  PROC DrawPart69()
    MoveL Offs(pOrigin,197.94,316.10,6.00),vTravel,z5,tPen\WObj:=wPaper;
    MoveL Offs(pOrigin,197.94,316.10,0.00),v60,z0,tPen\WObj:=wPaper;
    MoveL Offs(pOrigin,198.79,316.95,0.00),v40,z0,tPen\WObj:=wPaper;
    MoveL Offs(pOrigin,197.94,316.10,0.00),v40,fine,tPen\WObj:=wPaper;
    MoveL Offs(pOrigin,197.94,316.10,6.00),v60,z5,tPen\WObj:=wPaper;
    MoveL Offs(pOrigin,199.64,321.62,6.00),vTravel,z5,tPen\WObj:=wPaper;
    MoveL Offs(pOrigin,199.64,321.62,0.00),v60,z0,tPen\WObj:=wPaper;
    MoveL Offs(pOrigin,200.49,322.48,0.00),v40,z0,tPen\WObj:=wPaper;
    MoveL Offs(pOrigin,199.64,321.62,0.00),v40,fine,tPen\WObj:=wPaper;
    MoveL Offs(pOrigin,199.64,321.62,6.00),v60,z5,tPen\WObj:=wPaper;
    MoveL Offs(pOrigin,203.04,325.02,6.00),vTravel,z5,tPen\WObj:=wPaper;
    MoveL Offs(pOrigin,203.04,325.02,0.00),v60,z0,tPen\WObj:=wPaper;
    MoveL Offs(pOrigin,204.24,325.31,0.00),v40,z0,tPen\WObj:=wPaper;
    MoveL Offs(pOrigin,204.52,326.51,0.00),v40,z0,tPen\WObj:=wPaper;
    MoveL Offs(pOrigin,204.95,327.15,0.00),v40,z0,tPen\WObj:=wPaper;
    MoveL Offs(pOrigin,206.86,327.36,0.00),v40,fine,tPen\WObj:=wPaper;
    MoveL Offs(pOrigin,206.86,327.36,6.00),v60,z5,tPen\WObj:=wPaper;
    MoveL Offs(pOrigin,207.29,328.85,6.00),vTravel,z5,tPen\WObj:=wPaper;
    MoveL Offs(pOrigin,207.29,328.85,0.00),v60,z0,tPen\WObj:=wPaper;
    MoveL Offs(pOrigin,208.14,329.49,0.00),v40,z0,tPen\WObj:=wPaper;
    MoveL Offs(pOrigin,207.29,328.85,0.00),v40,fine,tPen\WObj:=wPaper;
    MoveL Offs(pOrigin,207.29,328.85,6.00),v60,z5,tPen\WObj:=wPaper;
    MoveL Offs(pOrigin,206.01,329.27,6.00),vTravel,z5,tPen\WObj:=wPaper;
    MoveL Offs(pOrigin,206.01,329.27,0.00),v60,z0,tPen\WObj:=wPaper;
    MoveL Offs(pOrigin,207.07,330.34,0.00),v40,z0,tPen\WObj:=wPaper;
    MoveL Offs(pOrigin,206.01,329.27,0.00),v40,z0,tPen\WObj:=wPaper;
    MoveL Offs(pOrigin,205.59,328.64,0.00),v40,z0,tPen\WObj:=wPaper;
    MoveL Offs(pOrigin,205.80,329.06,0.00),v40,z0,tPen\WObj:=wPaper;
    MoveL Offs(pOrigin,205.59,328.64,0.00),v40,fine,tPen\WObj:=wPaper;
    MoveL Offs(pOrigin,205.59,328.64,6.00),v60,z5,tPen\WObj:=wPaper;
    MoveL Offs(pOrigin,205.16,329.91,6.00),vTravel,z5,tPen\WObj:=wPaper;
    MoveL Offs(pOrigin,205.16,329.91,0.00),v60,z0,tPen\WObj:=wPaper;
    MoveL Offs(pOrigin,207.29,332.04,0.00),v40,z0,tPen\WObj:=wPaper;
    MoveL Offs(pOrigin,205.16,329.91,0.00),v40,fine,tPen\WObj:=wPaper;
    MoveL Offs(pOrigin,205.16,329.91,6.00),v60,z5,tPen\WObj:=wPaper;
    MoveL Offs(pOrigin,204.95,327.15,6.00),vTravel,z5,tPen\WObj:=wPaper;
    MoveL Offs(pOrigin,204.95,327.15,0.00),v60,z0,tPen\WObj:=wPaper;
    MoveL Offs(pOrigin,205.38,328.21,0.00),v40,z0,tPen\WObj:=wPaper;
    MoveL Offs(pOrigin,207.07,330.12,0.00),v40,z0,tPen\WObj:=wPaper;
    MoveL Offs(pOrigin,209.41,331.75,0.00),v40,z0,tPen\WObj:=wPaper;
    MoveL Offs(pOrigin,210.90,332.04,0.00),v40,z0,tPen\WObj:=wPaper;
    MoveL Offs(pOrigin,210.69,331.19,0.00),v40,z0,tPen\WObj:=wPaper;
    MoveL Offs(pOrigin,210.90,331.61,0.00),v40,z0,tPen\WObj:=wPaper;
    MoveL Offs(pOrigin,210.69,331.19,0.00),v40,fine,tPen\WObj:=wPaper;
    MoveL Offs(pOrigin,210.69,331.19,6.00),v60,z5,tPen\WObj:=wPaper;
    MoveL Offs(pOrigin,208.56,331.40,6.00),vTravel,z5,tPen\WObj:=wPaper;
    MoveL Offs(pOrigin,208.56,331.40,0.00),v60,z0,tPen\WObj:=wPaper;
    MoveL Offs(pOrigin,208.99,331.61,0.00),v40,z0,tPen\WObj:=wPaper;
    MoveL Offs(pOrigin,208.56,331.40,0.00),v40,z0,tPen\WObj:=wPaper;
    MoveL Offs(pOrigin,207.93,330.98,0.00),v40,z0,tPen\WObj:=wPaper;
    MoveL Offs(pOrigin,208.35,331.19,0.00),v40,z0,tPen\WObj:=wPaper;
    MoveL Offs(pOrigin,207.93,330.98,0.00),v40,fine,tPen\WObj:=wPaper;
    MoveL Offs(pOrigin,207.93,330.98,6.00),v60,z5,tPen\WObj:=wPaper;
    MoveL Offs(pOrigin,208.35,329.70,6.00),vTravel,z5,tPen\WObj:=wPaper;
    MoveL Offs(pOrigin,208.35,329.70,0.00),v60,z0,tPen\WObj:=wPaper;
    MoveL Offs(pOrigin,208.77,330.12,0.00),v40,z0,tPen\WObj:=wPaper;
    MoveL Offs(pOrigin,208.35,329.70,0.00),v40,fine,tPen\WObj:=wPaper;
    MoveL Offs(pOrigin,208.35,329.70,6.00),v60,z5,tPen\WObj:=wPaper;
    MoveL Offs(pOrigin,208.14,332.67,6.00),vTravel,z5,tPen\WObj:=wPaper;
    MoveL Offs(pOrigin,208.14,332.67,0.00),v60,z0,tPen\WObj:=wPaper;
    MoveL Offs(pOrigin,208.56,333.10,0.00),v40,z0,tPen\WObj:=wPaper;
    MoveL Offs(pOrigin,208.14,332.67,0.00),v40,fine,tPen\WObj:=wPaper;
    MoveL Offs(pOrigin,208.14,332.67,6.00),v60,z5,tPen\WObj:=wPaper;
    MoveL Offs(pOrigin,209.20,333.52,6.00),vTravel,z5,tPen\WObj:=wPaper;
    MoveL Offs(pOrigin,209.20,333.52,0.00),v60,z0,tPen\WObj:=wPaper;
    MoveL Offs(pOrigin,209.62,333.74,0.00),v40,z0,tPen\WObj:=wPaper;
    MoveL Offs(pOrigin,209.20,333.52,0.00),v40,fine,tPen\WObj:=wPaper;
    MoveL Offs(pOrigin,209.20,333.52,6.00),v60,z5,tPen\WObj:=wPaper;
    MoveL Offs(pOrigin,210.48,334.16,6.00),vTravel,z5,tPen\WObj:=wPaper;
    MoveL Offs(pOrigin,210.48,334.16,0.00),v60,z0,tPen\WObj:=wPaper;
    MoveL Offs(pOrigin,210.90,334.38,0.00),v40,z0,tPen\WObj:=wPaper;
    MoveL Offs(pOrigin,210.48,334.16,0.00),v40,fine,tPen\WObj:=wPaper;
    MoveL Offs(pOrigin,210.48,334.16,6.00),v60,z5,tPen\WObj:=wPaper;
    MoveL Offs(pOrigin,208.14,312.06,6.00),vTravel,z5,tPen\WObj:=wPaper;
    MoveL Offs(pOrigin,208.14,312.06,0.00),v60,z0,tPen\WObj:=wPaper;
    MoveL Offs(pOrigin,208.56,311.85,0.00),v40,z0,tPen\WObj:=wPaper;
    MoveL Offs(pOrigin,208.14,312.06,0.00),v40,fine,tPen\WObj:=wPaper;
    MoveL Offs(pOrigin,208.14,312.06,6.00),v60,z5,tPen\WObj:=wPaper;
    MoveL Offs(pOrigin,214.30,305.90,6.00),vTravel,z5,tPen\WObj:=wPaper;
    MoveL Offs(pOrigin,214.30,305.90,0.00),v60,z0,tPen\WObj:=wPaper;
    MoveL Offs(pOrigin,214.73,306.54,0.00),v40,z0,tPen\WObj:=wPaper;
    MoveL Offs(pOrigin,216.85,306.96,0.00),v40,z0,tPen\WObj:=wPaper;
    MoveL Offs(pOrigin,216.85,306.54,0.00),v40,z0,tPen\WObj:=wPaper;
    MoveL Offs(pOrigin,215.79,305.05,0.00),v40,z0,tPen\WObj:=wPaper;
    MoveL Offs(pOrigin,214.94,305.12,0.00),v40,z0,tPen\WObj:=wPaper;
    MoveL Offs(pOrigin,214.30,305.90,0.00),v40,fine,tPen\WObj:=wPaper;
    MoveL Offs(pOrigin,214.30,305.90,6.00),v60,z5,tPen\WObj:=wPaper;
    MoveL Offs(pOrigin,220.25,307.81,6.00),vTravel,z5,tPen\WObj:=wPaper;
    MoveL Offs(pOrigin,220.25,307.81,0.00),v60,z0,tPen\WObj:=wPaper;
    MoveL Offs(pOrigin,220.46,308.24,0.00),v40,z0,tPen\WObj:=wPaper;
    MoveL Offs(pOrigin,220.25,307.81,0.00),v40,fine,tPen\WObj:=wPaper;
    MoveL Offs(pOrigin,220.25,307.81,6.00),v60,z5,tPen\WObj:=wPaper;
    MoveL Offs(pOrigin,222.38,310.58,6.00),vTravel,z5,tPen\WObj:=wPaper;
    MoveL Offs(pOrigin,222.38,310.58,0.00),v60,z0,tPen\WObj:=wPaper;
    MoveL Offs(pOrigin,221.52,311.85,0.00),v40,fine,tPen\WObj:=wPaper;
    MoveL Offs(pOrigin,221.52,311.85,6.00),v60,z5,tPen\WObj:=wPaper;
    MoveL Offs(pOrigin,221.31,313.34,6.00),vTravel,z5,tPen\WObj:=wPaper;
    MoveL Offs(pOrigin,221.31,313.34,0.00),v60,z0,tPen\WObj:=wPaper;
    MoveL Offs(pOrigin,221.52,312.27,0.00),v40,z0,tPen\WObj:=wPaper;
    MoveL Offs(pOrigin,221.10,311.92,0.00),v40,z0,tPen\WObj:=wPaper;
    MoveL Offs(pOrigin,220.46,312.13,0.00),v40,z0,tPen\WObj:=wPaper;
    MoveL Offs(pOrigin,219.61,313.34,0.00),v40,fine,tPen\WObj:=wPaper;
    MoveL Offs(pOrigin,219.61,313.34,6.00),v60,z5,tPen\WObj:=wPaper;
    MoveL Offs(pOrigin,209.84,301.01,6.00),vTravel,z5,tPen\WObj:=wPaper;
    MoveL Offs(pOrigin,209.84,301.01,0.00),v60,z0,tPen\WObj:=wPaper;
    MoveL Offs(pOrigin,209.34,298.89,0.00),v40,z0,tPen\WObj:=wPaper;
    MoveL Offs(pOrigin,207.50,296.76,0.00),v40,z0,tPen\WObj:=wPaper;
    MoveL Offs(pOrigin,207.93,296.98,0.00),v40,z0,tPen\WObj:=wPaper;
    MoveL Offs(pOrigin,208.35,297.40,0.00),v40,z0,tPen\WObj:=wPaper;
    MoveL Offs(pOrigin,207.93,296.98,0.00),v40,fine,tPen\WObj:=wPaper;
    MoveL Offs(pOrigin,207.93,296.98,6.00),v60,z5,tPen\WObj:=wPaper;
    MoveL Offs(pOrigin,209.20,266.38,6.00),vTravel,z5,tPen\WObj:=wPaper;
    MoveL Offs(pOrigin,209.20,266.38,0.00),v60,z0,tPen\WObj:=wPaper;
    MoveL Offs(pOrigin,208.14,266.16,0.00),v40,z0,tPen\WObj:=wPaper;
    MoveL Offs(pOrigin,207.50,265.31,0.00),v40,fine,tPen\WObj:=wPaper;
    MoveL Offs(pOrigin,207.50,265.31,6.00),v60,z5,tPen\WObj:=wPaper;
    MoveL Offs(pOrigin,207.29,260.85,6.00),vTravel,z5,tPen\WObj:=wPaper;
    MoveL Offs(pOrigin,207.29,260.85,0.00),v60,z0,tPen\WObj:=wPaper;
    MoveL Offs(pOrigin,207.93,260.00,0.00),v40,z0,tPen\WObj:=wPaper;
    MoveL Offs(pOrigin,207.93,258.94,0.00),v40,z0,tPen\WObj:=wPaper;
  ENDPROC

  PROC DrawPart70()
    MoveL Offs(pOrigin,207.93,258.94,0.00),v40,z0,tPen\WObj:=wPaper;
    MoveL Offs(pOrigin,208.07,258.30,0.00),v40,z0,tPen\WObj:=wPaper;
    MoveL Offs(pOrigin,207.07,257.02,0.00),v40,z0,tPen\WObj:=wPaper;
    MoveL Offs(pOrigin,207.29,251.71,0.00),v40,z0,tPen\WObj:=wPaper;
    MoveL Offs(pOrigin,207.07,248.95,0.00),v40,z0,tPen\WObj:=wPaper;
    MoveL Offs(pOrigin,206.44,248.17,0.00),v40,z0,tPen\WObj:=wPaper;
    MoveL Offs(pOrigin,205.66,248.31,0.00),v40,z0,tPen\WObj:=wPaper;
    MoveL Offs(pOrigin,205.38,250.23,0.00),v40,z0,tPen\WObj:=wPaper;
    MoveL Offs(pOrigin,205.80,250.65,0.00),v40,z0,tPen\WObj:=wPaper;
    MoveL Offs(pOrigin,205.02,250.44,0.00),v40,z0,tPen\WObj:=wPaper;
    MoveL Offs(pOrigin,204.38,252.14,0.00),v40,z0,tPen\WObj:=wPaper;
    MoveL Offs(pOrigin,203.39,257.02,0.00),v40,z0,tPen\WObj:=wPaper;
    MoveL Offs(pOrigin,203.68,258.09,0.00),v40,z0,tPen\WObj:=wPaper;
    MoveL Offs(pOrigin,203.46,259.36,0.00),v40,z0,tPen\WObj:=wPaper;
    MoveL Offs(pOrigin,202.90,260.00,0.00),v40,z0,tPen\WObj:=wPaper;
    MoveL Offs(pOrigin,202.54,261.70,0.00),v40,z0,tPen\WObj:=wPaper;
    MoveL Offs(pOrigin,201.98,261.91,0.00),v40,z0,tPen\WObj:=wPaper;
    MoveL Offs(pOrigin,201.98,261.91,0.00),v40,z0,tPen\WObj:=wPaper;
    MoveL Offs(pOrigin,201.69,260.00,0.00),v40,z0,tPen\WObj:=wPaper;
    MoveL Offs(pOrigin,200.91,259.79,0.00),v40,z0,tPen\WObj:=wPaper;
    MoveL Offs(pOrigin,201.98,259.79,0.00),v40,z0,tPen\WObj:=wPaper;
    MoveL Offs(pOrigin,202.12,258.51,0.00),v40,z0,tPen\WObj:=wPaper;
    MoveL Offs(pOrigin,203.25,257.45,0.00),v40,fine,tPen\WObj:=wPaper;
    MoveL Offs(pOrigin,203.25,257.45,6.00),v60,z5,tPen\WObj:=wPaper;
    MoveL Offs(pOrigin,201.55,256.81,6.00),vTravel,z5,tPen\WObj:=wPaper;
    MoveL Offs(pOrigin,201.55,256.81,0.00),v60,z0,tPen\WObj:=wPaper;
    MoveL Offs(pOrigin,201.12,249.59,0.00),v40,fine,tPen\WObj:=wPaper;
    MoveL Offs(pOrigin,201.12,249.59,6.00),v60,z5,tPen\WObj:=wPaper;
    MoveL Offs(pOrigin,198.57,248.74,6.00),vTravel,z5,tPen\WObj:=wPaper;
    MoveL Offs(pOrigin,198.57,248.74,0.00),v60,z0,tPen\WObj:=wPaper;
    MoveL Offs(pOrigin,198.15,249.38,0.00),v40,z0,tPen\WObj:=wPaper;
    MoveL Offs(pOrigin,198.57,248.74,0.00),v40,fine,tPen\WObj:=wPaper;
    MoveL Offs(pOrigin,198.57,248.74,6.00),v60,z5,tPen\WObj:=wPaper;
    MoveL Offs(pOrigin,197.73,247.68,6.00),vTravel,z5,tPen\WObj:=wPaper;
    MoveL Offs(pOrigin,197.73,247.68,0.00),v60,z0,tPen\WObj:=wPaper;
    MoveL Offs(pOrigin,197.30,248.31,0.00),v40,z0,tPen\WObj:=wPaper;
    MoveL Offs(pOrigin,197.73,247.68,0.00),v40,fine,tPen\WObj:=wPaper;
    MoveL Offs(pOrigin,197.73,247.68,6.00),v60,z5,tPen\WObj:=wPaper;
    MoveL Offs(pOrigin,198.79,245.98,6.00),vTravel,z5,tPen\WObj:=wPaper;
    MoveL Offs(pOrigin,198.79,245.98,0.00),v60,z0,tPen\WObj:=wPaper;
    MoveL Offs(pOrigin,198.36,246.61,0.00),v40,z0,tPen\WObj:=wPaper;
    MoveL Offs(pOrigin,198.79,245.98,0.00),v40,fine,tPen\WObj:=wPaper;
    MoveL Offs(pOrigin,198.79,245.98,6.00),v60,z5,tPen\WObj:=wPaper;
    MoveL Offs(pOrigin,199.64,247.04,6.00),vTravel,z5,tPen\WObj:=wPaper;
    MoveL Offs(pOrigin,199.64,247.04,0.00),v60,z0,tPen\WObj:=wPaper;
    MoveL Offs(pOrigin,199.43,247.46,0.00),v40,z0,tPen\WObj:=wPaper;
    MoveL Offs(pOrigin,199.64,247.04,0.00),v40,fine,tPen\WObj:=wPaper;
    MoveL Offs(pOrigin,199.64,247.04,6.00),v60,z5,tPen\WObj:=wPaper;
    MoveL Offs(pOrigin,197.73,250.01,6.00),vTravel,z5,tPen\WObj:=wPaper;
    MoveL Offs(pOrigin,197.73,250.01,0.00),v60,z0,tPen\WObj:=wPaper;
    MoveL Offs(pOrigin,197.51,250.44,0.00),v40,z0,tPen\WObj:=wPaper;
    MoveL Offs(pOrigin,197.73,250.01,0.00),v40,z0,tPen\WObj:=wPaper;
    MoveL Offs(pOrigin,197.30,250.86,0.00),v40,z0,tPen\WObj:=wPaper;
    MoveL Offs(pOrigin,197.09,251.29,0.00),v40,z0,tPen\WObj:=wPaper;
    MoveL Offs(pOrigin,197.30,250.86,0.00),v40,fine,tPen\WObj:=wPaper;
    MoveL Offs(pOrigin,197.30,250.86,6.00),v60,z5,tPen\WObj:=wPaper;
    MoveL Offs(pOrigin,196.24,249.80,6.00),vTravel,z5,tPen\WObj:=wPaper;
    MoveL Offs(pOrigin,196.24,249.80,0.00),v60,z0,tPen\WObj:=wPaper;
    MoveL Offs(pOrigin,196.02,250.23,0.00),v40,z0,tPen\WObj:=wPaper;
    MoveL Offs(pOrigin,196.24,249.80,0.00),v40,fine,tPen\WObj:=wPaper;
    MoveL Offs(pOrigin,196.24,249.80,6.00),v60,z5,tPen\WObj:=wPaper;
    MoveL Offs(pOrigin,205.59,248.10,6.00),vTravel,z5,tPen\WObj:=wPaper;
    MoveL Offs(pOrigin,205.59,248.10,0.00),v60,z0,tPen\WObj:=wPaper;
    MoveL Offs(pOrigin,204.95,247.04,0.00),v40,z0,tPen\WObj:=wPaper;
    MoveL Offs(pOrigin,204.81,245.34,0.00),v40,z0,tPen\WObj:=wPaper;
    MoveL Offs(pOrigin,205.09,243.85,0.00),v40,z0,tPen\WObj:=wPaper;
    MoveL Offs(pOrigin,205.59,243.21,0.00),v40,z0,tPen\WObj:=wPaper;
    MoveL Offs(pOrigin,205.59,243.21,0.00),v40,z0,tPen\WObj:=wPaper;
    MoveL Offs(pOrigin,205.80,241.94,0.00),v40,z0,tPen\WObj:=wPaper;
    MoveL Offs(pOrigin,206.65,241.51,0.00),v40,z0,tPen\WObj:=wPaper;
    MoveL Offs(pOrigin,206.65,241.51,0.00),v40,z0,tPen\WObj:=wPaper;
    MoveL Offs(pOrigin,206.86,242.79,0.00),v40,z0,tPen\WObj:=wPaper;
    MoveL Offs(pOrigin,206.44,243.21,0.00),v40,z0,tPen\WObj:=wPaper;
    MoveL Offs(pOrigin,206.44,243.21,0.00),v40,z0,tPen\WObj:=wPaper;
    MoveL Offs(pOrigin,206.86,245.98,0.00),v40,z0,tPen\WObj:=wPaper;
    MoveL Offs(pOrigin,206.65,248.10,0.00),v40,fine,tPen\WObj:=wPaper;
    MoveL Offs(pOrigin,206.65,248.10,6.00),v60,z5,tPen\WObj:=wPaper;
    MoveL Offs(pOrigin,207.29,257.24,6.00),vTravel,z5,tPen\WObj:=wPaper;
    MoveL Offs(pOrigin,207.29,257.24,0.00),v60,z0,tPen\WObj:=wPaper;
    MoveL Offs(pOrigin,207.71,257.45,0.00),v40,z0,tPen\WObj:=wPaper;
    MoveL Offs(pOrigin,208.07,257.24,0.00),v40,z0,tPen\WObj:=wPaper;
    MoveL Offs(pOrigin,209.34,253.41,0.00),v40,z0,tPen\WObj:=wPaper;
    MoveL Offs(pOrigin,210.90,251.07,0.00),v40,z0,tPen\WObj:=wPaper;
    MoveL Offs(pOrigin,211.96,250.30,0.00),v40,z0,tPen\WObj:=wPaper;
    MoveL Offs(pOrigin,214.94,249.59,0.00),v40,z0,tPen\WObj:=wPaper;
    MoveL Offs(pOrigin,223.65,249.80,0.00),v40,z0,tPen\WObj:=wPaper;
    MoveL Offs(pOrigin,230.45,251.07,0.00),v40,z0,tPen\WObj:=wPaper;
    MoveL Offs(pOrigin,232.79,251.85,0.00),v40,z0,tPen\WObj:=wPaper;
    MoveL Offs(pOrigin,234.91,253.62,0.00),v40,z0,tPen\WObj:=wPaper;
    MoveL Offs(pOrigin,235.55,254.90,0.00),v40,fine,tPen\WObj:=wPaper;
    MoveL Offs(pOrigin,235.55,254.90,6.00),v60,z5,tPen\WObj:=wPaper;
    MoveL Offs(pOrigin,236.19,256.39,6.00),vTravel,z5,tPen\WObj:=wPaper;
    MoveL Offs(pOrigin,236.19,256.39,0.00),v60,z0,tPen\WObj:=wPaper;
    MoveL Offs(pOrigin,236.19,257.24,0.00),v40,z0,tPen\WObj:=wPaper;
    MoveL Offs(pOrigin,236.82,257.88,0.00),v40,z0,tPen\WObj:=wPaper;
    MoveL Offs(pOrigin,236.82,257.88,0.00),v40,z0,tPen\WObj:=wPaper;
    MoveL Offs(pOrigin,237.68,257.02,0.00),v40,z0,tPen\WObj:=wPaper;
    MoveL Offs(pOrigin,237.60,256.17,0.00),v40,z0,tPen\WObj:=wPaper;
    MoveL Offs(pOrigin,237.04,255.75,0.00),v40,z0,tPen\WObj:=wPaper;
    MoveL Offs(pOrigin,237.04,255.75,0.00),v40,z0,tPen\WObj:=wPaper;
    MoveL Offs(pOrigin,236.19,256.39,0.00),v40,z0,tPen\WObj:=wPaper;
    MoveL Offs(pOrigin,236.19,256.39,0.00),v40,z0,tPen\WObj:=wPaper;
    MoveL Offs(pOrigin,235.69,255.96,0.00),v40,z0,tPen\WObj:=wPaper;
    MoveL Offs(pOrigin,235.62,255.11,0.00),v40,z0,tPen\WObj:=wPaper;
    MoveL Offs(pOrigin,236.40,255.18,0.00),v40,z0,tPen\WObj:=wPaper;
    MoveL Offs(pOrigin,237.04,255.75,0.00),v40,fine,tPen\WObj:=wPaper;
    MoveL Offs(pOrigin,237.04,255.75,6.00),v60,z5,tPen\WObj:=wPaper;
    MoveL Offs(pOrigin,236.82,259.58,6.00),vTravel,z5,tPen\WObj:=wPaper;
    MoveL Offs(pOrigin,236.82,259.58,0.00),v60,z0,tPen\WObj:=wPaper;
    MoveL Offs(pOrigin,236.75,258.51,0.00),v40,z0,tPen\WObj:=wPaper;
    MoveL Offs(pOrigin,235.98,258.09,0.00),v40,z0,tPen\WObj:=wPaper;
    MoveL Offs(pOrigin,234.49,259.58,0.00),v40,z0,tPen\WObj:=wPaper;
    MoveL Offs(pOrigin,234.49,259.58,0.00),v40,z0,tPen\WObj:=wPaper;
    MoveL Offs(pOrigin,235.12,260.21,0.00),v40,z0,tPen\WObj:=wPaper;
    MoveL Offs(pOrigin,235.12,260.21,0.00),v40,z0,tPen\WObj:=wPaper;
    MoveL Offs(pOrigin,235.12,260.00,0.00),v40,z0,tPen\WObj:=wPaper;
    MoveL Offs(pOrigin,236.19,260.21,0.00),v40,z0,tPen\WObj:=wPaper;
    MoveL Offs(pOrigin,236.82,259.58,0.00),v40,z0,tPen\WObj:=wPaper;
    MoveL Offs(pOrigin,236.82,259.58,0.00),v40,z0,tPen\WObj:=wPaper;
    MoveL Offs(pOrigin,237.04,260.85,0.00),v40,z0,tPen\WObj:=wPaper;
  ENDPROC

  PROC DrawPart71()
    MoveL Offs(pOrigin,237.04,260.85,0.00),v40,z0,tPen\WObj:=wPaper;
    MoveL Offs(pOrigin,238.31,262.12,0.00),v40,z0,tPen\WObj:=wPaper;
    MoveL Offs(pOrigin,238.24,262.98,0.00),v40,z0,tPen\WObj:=wPaper;
    MoveL Offs(pOrigin,237.25,263.83,0.00),v40,z0,tPen\WObj:=wPaper;
    MoveL Offs(pOrigin,237.25,263.83,0.00),v40,z0,tPen\WObj:=wPaper;
    MoveL Offs(pOrigin,238.10,265.31,0.00),v40,z0,tPen\WObj:=wPaper;
    MoveL Offs(pOrigin,240.23,266.16,0.00),v40,z0,tPen\WObj:=wPaper;
    MoveL Offs(pOrigin,243.41,266.38,0.00),v40,z0,tPen\WObj:=wPaper;
    MoveL Offs(pOrigin,244.69,266.16,0.00),v40,fine,tPen\WObj:=wPaper;
    MoveL Offs(pOrigin,244.69,266.16,6.00),v60,z5,tPen\WObj:=wPaper;
    MoveL Offs(pOrigin,244.69,267.86,6.00),vTravel,z5,tPen\WObj:=wPaper;
    MoveL Offs(pOrigin,244.69,267.86,0.00),v60,z0,tPen\WObj:=wPaper;
    MoveL Offs(pOrigin,245.75,267.65,0.00),v40,z0,tPen\WObj:=wPaper;
    MoveL Offs(pOrigin,245.75,267.86,0.00),v40,z0,tPen\WObj:=wPaper;
    MoveL Offs(pOrigin,246.60,267.86,0.00),v40,z0,tPen\WObj:=wPaper;
    MoveL Offs(pOrigin,245.96,267.93,0.00),v40,z0,tPen\WObj:=wPaper;
    MoveL Offs(pOrigin,245.75,268.50,0.00),v40,z0,tPen\WObj:=wPaper;
    MoveL Offs(pOrigin,246.81,269.14,0.00),v40,fine,tPen\WObj:=wPaper;
    MoveL Offs(pOrigin,246.81,269.14,6.00),v60,z5,tPen\WObj:=wPaper;
    MoveL Offs(pOrigin,247.24,270.41,6.00),vTravel,z5,tPen\WObj:=wPaper;
    MoveL Offs(pOrigin,247.24,270.41,0.00),v60,z0,tPen\WObj:=wPaper;
    MoveL Offs(pOrigin,248.73,270.62,0.00),v40,fine,tPen\WObj:=wPaper;
    MoveL Offs(pOrigin,248.73,270.62,6.00),v60,z5,tPen\WObj:=wPaper;
    MoveL Offs(pOrigin,247.24,270.41,6.00),vTravel,z5,tPen\WObj:=wPaper;
    MoveL Offs(pOrigin,247.24,270.41,0.00),v60,z0,tPen\WObj:=wPaper;
    MoveL Offs(pOrigin,246.18,271.90,0.00),v40,z0,tPen\WObj:=wPaper;
    MoveL Offs(pOrigin,246.25,272.54,0.00),v40,z0,tPen\WObj:=wPaper;
    MoveL Offs(pOrigin,246.81,272.96,0.00),v40,fine,tPen\WObj:=wPaper;
    MoveL Offs(pOrigin,246.81,272.96,6.00),v60,z5,tPen\WObj:=wPaper;
    MoveL Offs(pOrigin,245.11,270.20,6.00),vTravel,z5,tPen\WObj:=wPaper;
    MoveL Offs(pOrigin,245.11,270.20,0.00),v60,z0,tPen\WObj:=wPaper;
    MoveL Offs(pOrigin,243.98,271.26,0.00),v40,z0,tPen\WObj:=wPaper;
    MoveL Offs(pOrigin,243.13,273.17,0.00),v40,z0,tPen\WObj:=wPaper;
    MoveL Offs(pOrigin,242.14,277.64,0.00),v40,fine,tPen\WObj:=wPaper;
    MoveL Offs(pOrigin,242.14,277.64,6.00),v60,z5,tPen\WObj:=wPaper;
    MoveL Offs(pOrigin,237.46,267.01,6.00),vTravel,z5,tPen\WObj:=wPaper;
    MoveL Offs(pOrigin,237.46,267.01,0.00),v60,z0,tPen\WObj:=wPaper;
    MoveL Offs(pOrigin,237.04,266.23,0.00),v40,z0,tPen\WObj:=wPaper;
    MoveL Offs(pOrigin,236.40,266.23,0.00),v40,z0,tPen\WObj:=wPaper;
    MoveL Offs(pOrigin,235.69,267.01,0.00),v40,z0,tPen\WObj:=wPaper;
    MoveL Offs(pOrigin,236.40,267.44,0.00),v40,fine,tPen\WObj:=wPaper;
    MoveL Offs(pOrigin,236.40,267.44,6.00),v60,z5,tPen\WObj:=wPaper;
    MoveL Offs(pOrigin,235.34,265.52,6.00),vTravel,z5,tPen\WObj:=wPaper;
    MoveL Offs(pOrigin,235.34,265.52,0.00),v60,z0,tPen\WObj:=wPaper;
    MoveL Offs(pOrigin,235.98,264.67,0.00),v40,z0,tPen\WObj:=wPaper;
    MoveL Offs(pOrigin,237.25,263.83,0.00),v40,z0,tPen\WObj:=wPaper;
    MoveL Offs(pOrigin,236.82,263.83,0.00),v40,z0,tPen\WObj:=wPaper;
    MoveL Offs(pOrigin,236.19,262.55,0.00),v40,z0,tPen\WObj:=wPaper;
    MoveL Offs(pOrigin,235.34,262.34,0.00),v40,z0,tPen\WObj:=wPaper;
    MoveL Offs(pOrigin,235.34,262.34,0.00),v40,z0,tPen\WObj:=wPaper;
    MoveL Offs(pOrigin,234.91,261.27,0.00),v40,z0,tPen\WObj:=wPaper;
    MoveL Offs(pOrigin,235.12,260.21,0.00),v40,z0,tPen\WObj:=wPaper;
    MoveL Offs(pOrigin,234.49,259.58,0.00),v40,z0,tPen\WObj:=wPaper;
    MoveL Offs(pOrigin,233.21,259.50,0.00),v40,z0,tPen\WObj:=wPaper;
    MoveL Offs(pOrigin,232.72,258.09,0.00),v40,z0,tPen\WObj:=wPaper;
    MoveL Offs(pOrigin,231.30,256.60,0.00),v40,z0,tPen\WObj:=wPaper;
    MoveL Offs(pOrigin,227.05,254.26,0.00),v40,fine,tPen\WObj:=wPaper;
    MoveL Offs(pOrigin,227.05,254.26,6.00),v60,z5,tPen\WObj:=wPaper;
    MoveL Offs(pOrigin,226.41,259.15,6.00),vTravel,z5,tPen\WObj:=wPaper;
    MoveL Offs(pOrigin,226.41,259.15,0.00),v60,z0,tPen\WObj:=wPaper;
    MoveL Offs(pOrigin,223.65,258.94,0.00),v40,z0,tPen\WObj:=wPaper;
    MoveL Offs(pOrigin,223.23,259.15,0.00),v40,z0,tPen\WObj:=wPaper;
    MoveL Offs(pOrigin,222.87,260.00,0.00),v40,z0,tPen\WObj:=wPaper;
    MoveL Offs(pOrigin,224.07,260.85,0.00),v40,z0,tPen\WObj:=wPaper;
    MoveL Offs(pOrigin,224.07,260.85,0.00),v40,z0,tPen\WObj:=wPaper;
    MoveL Offs(pOrigin,224.29,261.49,0.00),v40,z0,tPen\WObj:=wPaper;
    MoveL Offs(pOrigin,224.71,261.70,0.00),v40,z0,tPen\WObj:=wPaper;
    MoveL Offs(pOrigin,225.56,261.63,0.00),v40,z0,tPen\WObj:=wPaper;
    MoveL Offs(pOrigin,226.20,261.06,0.00),v40,z0,tPen\WObj:=wPaper;
    MoveL Offs(pOrigin,227.05,261.06,0.00),v40,z0,tPen\WObj:=wPaper;
    MoveL Offs(pOrigin,227.48,260.64,0.00),v40,z0,tPen\WObj:=wPaper;
    MoveL Offs(pOrigin,228.32,260.64,0.00),v40,z0,tPen\WObj:=wPaper;
    MoveL Offs(pOrigin,228.96,261.27,0.00),v40,z0,tPen\WObj:=wPaper;
    MoveL Offs(pOrigin,228.96,261.91,0.00),v40,z0,tPen\WObj:=wPaper;
    MoveL Offs(pOrigin,229.03,261.49,0.00),v40,z0,tPen\WObj:=wPaper;
    MoveL Offs(pOrigin,229.60,261.27,0.00),v40,z0,tPen\WObj:=wPaper;
    MoveL Offs(pOrigin,230.88,261.63,0.00),v40,z0,tPen\WObj:=wPaper;
    MoveL Offs(pOrigin,231.51,262.34,0.00),v40,z0,tPen\WObj:=wPaper;
    MoveL Offs(pOrigin,231.30,261.70,0.00),v40,z0,tPen\WObj:=wPaper;
    MoveL Offs(pOrigin,232.36,261.27,0.00),v40,z0,tPen\WObj:=wPaper;
    MoveL Offs(pOrigin,233.21,261.49,0.00),v40,z0,tPen\WObj:=wPaper;
    MoveL Offs(pOrigin,233.21,261.49,0.00),v40,z0,tPen\WObj:=wPaper;
    MoveL Offs(pOrigin,234.91,261.49,0.00),v40,fine,tPen\WObj:=wPaper;
    MoveL Offs(pOrigin,234.91,261.49,6.00),v60,z5,tPen\WObj:=wPaper;
    MoveL Offs(pOrigin,236.19,262.34,6.00),vTravel,z5,tPen\WObj:=wPaper;
    MoveL Offs(pOrigin,236.19,262.34,0.00),v60,z0,tPen\WObj:=wPaper;
    MoveL Offs(pOrigin,237.04,260.85,0.00),v40,fine,tPen\WObj:=wPaper;
    MoveL Offs(pOrigin,237.04,260.85,6.00),v60,z5,tPen\WObj:=wPaper;
    MoveL Offs(pOrigin,233.00,259.58,6.00),vTravel,z5,tPen\WObj:=wPaper;
    MoveL Offs(pOrigin,233.00,259.58,0.00),v60,z0,tPen\WObj:=wPaper;
    MoveL Offs(pOrigin,231.51,259.29,0.00),v40,z0,tPen\WObj:=wPaper;
    MoveL Offs(pOrigin,227.26,257.31,0.00),v40,z0,tPen\WObj:=wPaper;
    MoveL Offs(pOrigin,224.50,256.60,0.00),v40,z0,tPen\WObj:=wPaper;
    MoveL Offs(pOrigin,223.23,256.60,0.00),v40,z0,tPen\WObj:=wPaper;
    MoveL Offs(pOrigin,222.16,255.96,0.00),v40,fine,tPen\WObj:=wPaper;
    MoveL Offs(pOrigin,222.16,255.96,6.00),v60,z5,tPen\WObj:=wPaper;
    MoveL Offs(pOrigin,221.74,257.24,6.00),vTravel,z5,tPen\WObj:=wPaper;
    MoveL Offs(pOrigin,221.74,257.24,0.00),v60,z0,tPen\WObj:=wPaper;
    MoveL Offs(pOrigin,219.19,257.45,0.00),v40,fine,tPen\WObj:=wPaper;
    MoveL Offs(pOrigin,219.19,257.45,6.00),v60,z5,tPen\WObj:=wPaper;
    MoveL Offs(pOrigin,213.24,263.40,6.00),vTravel,z5,tPen\WObj:=wPaper;
    MoveL Offs(pOrigin,213.24,263.40,0.00),v60,z0,tPen\WObj:=wPaper;
    MoveL Offs(pOrigin,213.10,264.89,0.00),v40,z0,tPen\WObj:=wPaper;
    MoveL Offs(pOrigin,214.51,266.59,0.00),v40,z0,tPen\WObj:=wPaper;
    MoveL Offs(pOrigin,219.19,267.86,0.00),v40,z0,tPen\WObj:=wPaper;
    MoveL Offs(pOrigin,219.19,267.86,0.00),v40,z0,tPen\WObj:=wPaper;
    MoveL Offs(pOrigin,220.89,268.08,0.00),v40,z0,tPen\WObj:=wPaper;
    MoveL Offs(pOrigin,221.74,267.86,0.00),v40,fine,tPen\WObj:=wPaper;
    MoveL Offs(pOrigin,221.74,267.86,6.00),v60,z5,tPen\WObj:=wPaper;
    MoveL Offs(pOrigin,233.21,267.44,6.00),vTravel,z5,tPen\WObj:=wPaper;
    MoveL Offs(pOrigin,233.21,267.44,0.00),v60,z0,tPen\WObj:=wPaper;
    MoveL Offs(pOrigin,233.85,268.08,0.00),v40,fine,tPen\WObj:=wPaper;
    MoveL Offs(pOrigin,233.85,268.08,6.00),v60,z5,tPen\WObj:=wPaper;
    MoveL Offs(pOrigin,252.12,268.29,6.00),vTravel,z5,tPen\WObj:=wPaper;
    MoveL Offs(pOrigin,252.12,268.29,0.00),v60,z0,tPen\WObj:=wPaper;
    MoveL Offs(pOrigin,252.55,268.71,0.00),v40,z0,tPen\WObj:=wPaper;
    MoveL Offs(pOrigin,252.12,268.29,0.00),v40,fine,tPen\WObj:=wPaper;
    MoveL Offs(pOrigin,252.12,268.29,6.00),v60,z5,tPen\WObj:=wPaper;
    MoveL Offs(pOrigin,255.95,269.35,6.00),vTravel,z5,tPen\WObj:=wPaper;
    MoveL Offs(pOrigin,255.95,269.35,0.00),v60,z0,tPen\WObj:=wPaper;
  ENDPROC

  PROC DrawPart72()
    MoveL Offs(pOrigin,257.44,269.99,0.00),v40,z0,tPen\WObj:=wPaper;
    MoveL Offs(pOrigin,259.14,269.77,0.00),v40,fine,tPen\WObj:=wPaper;
    MoveL Offs(pOrigin,259.14,269.77,6.00),v60,z5,tPen\WObj:=wPaper;
    MoveL Offs(pOrigin,276.35,263.83,6.00),vTravel,z5,tPen\WObj:=wPaper;
    MoveL Offs(pOrigin,276.35,263.83,0.00),v60,z0,tPen\WObj:=wPaper;
    MoveL Offs(pOrigin,275.92,263.40,0.00),v40,z0,tPen\WObj:=wPaper;
    MoveL Offs(pOrigin,276.14,262.34,0.00),v40,z0,tPen\WObj:=wPaper;
    MoveL Offs(pOrigin,276.14,261.91,0.00),v40,z0,tPen\WObj:=wPaper;
    MoveL Offs(pOrigin,275.71,261.49,0.00),v40,z0,tPen\WObj:=wPaper;
    MoveL Offs(pOrigin,275.92,260.64,0.00),v40,fine,tPen\WObj:=wPaper;
    MoveL Offs(pOrigin,275.92,260.64,6.00),v60,z5,tPen\WObj:=wPaper;
    MoveL Offs(pOrigin,279.75,272.75,6.00),vTravel,z5,tPen\WObj:=wPaper;
    MoveL Offs(pOrigin,279.75,272.75,0.00),v60,z0,tPen\WObj:=wPaper;
    MoveL Offs(pOrigin,280.39,273.17,0.00),v40,z0,tPen\WObj:=wPaper;
    MoveL Offs(pOrigin,282.09,273.17,0.00),v40,fine,tPen\WObj:=wPaper;
    MoveL Offs(pOrigin,282.09,273.17,6.00),v60,z5,tPen\WObj:=wPaper;
    MoveL Offs(pOrigin,280.39,279.12,6.00),vTravel,z5,tPen\WObj:=wPaper;
    MoveL Offs(pOrigin,280.39,279.12,0.00),v60,z0,tPen\WObj:=wPaper;
    MoveL Offs(pOrigin,279.61,279.41,0.00),v40,z0,tPen\WObj:=wPaper;
    MoveL Offs(pOrigin,279.33,280.19,0.00),v40,z0,tPen\WObj:=wPaper;
    MoveL Offs(pOrigin,279.96,280.83,0.00),v40,fine,tPen\WObj:=wPaper;
    MoveL Offs(pOrigin,279.96,280.83,6.00),v60,z5,tPen\WObj:=wPaper;
    MoveL Offs(pOrigin,291.44,271.48,6.00),vTravel,z5,tPen\WObj:=wPaper;
    MoveL Offs(pOrigin,291.44,271.48,0.00),v60,z0,tPen\WObj:=wPaper;
    MoveL Offs(pOrigin,291.44,270.41,0.00),v40,z0,tPen\WObj:=wPaper;
    MoveL Offs(pOrigin,290.38,269.99,0.00),v40,z0,tPen\WObj:=wPaper;
    MoveL Offs(pOrigin,290.38,269.99,0.00),v40,z0,tPen\WObj:=wPaper;
    MoveL Offs(pOrigin,290.16,269.42,0.00),v40,z0,tPen\WObj:=wPaper;
    MoveL Offs(pOrigin,289.10,268.92,0.00),v40,z0,tPen\WObj:=wPaper;
    MoveL Offs(pOrigin,289.17,268.36,0.00),v40,z0,tPen\WObj:=wPaper;
    MoveL Offs(pOrigin,289.95,268.29,0.00),v40,z0,tPen\WObj:=wPaper;
    MoveL Offs(pOrigin,289.95,268.29,0.00),v40,z0,tPen\WObj:=wPaper;
    MoveL Offs(pOrigin,290.38,269.35,0.00),v40,z0,tPen\WObj:=wPaper;
    MoveL Offs(pOrigin,290.38,269.99,0.00),v40,z0,tPen\WObj:=wPaper;
    MoveL Offs(pOrigin,290.16,270.41,0.00),v40,z0,tPen\WObj:=wPaper;
    MoveL Offs(pOrigin,290.38,271.05,0.00),v40,z0,tPen\WObj:=wPaper;
    MoveL Offs(pOrigin,291.44,271.48,0.00),v40,fine,tPen\WObj:=wPaper;
    MoveL Offs(pOrigin,291.44,271.48,6.00),v60,z5,tPen\WObj:=wPaper;
    MoveL Offs(pOrigin,293.56,269.77,6.00),vTravel,z5,tPen\WObj:=wPaper;
    MoveL Offs(pOrigin,293.56,269.77,0.00),v60,z0,tPen\WObj:=wPaper;
    MoveL Offs(pOrigin,294.20,270.41,0.00),v40,z0,tPen\WObj:=wPaper;
    MoveL Offs(pOrigin,293.56,269.77,0.00),v40,fine,tPen\WObj:=wPaper;
    MoveL Offs(pOrigin,293.56,269.77,6.00),v60,z5,tPen\WObj:=wPaper;
    MoveL Offs(pOrigin,290.80,267.23,6.00),vTravel,z5,tPen\WObj:=wPaper;
    MoveL Offs(pOrigin,290.80,267.23,0.00),v60,z0,tPen\WObj:=wPaper;
    MoveL Offs(pOrigin,289.95,267.86,0.00),v40,z0,tPen\WObj:=wPaper;
    MoveL Offs(pOrigin,289.95,268.29,0.00),v40,fine,tPen\WObj:=wPaper;
    MoveL Offs(pOrigin,289.95,268.29,6.00),v60,z5,tPen\WObj:=wPaper;
    MoveL Offs(pOrigin,264.66,312.27,6.00),vTravel,z5,tPen\WObj:=wPaper;
    MoveL Offs(pOrigin,264.66,312.27,0.00),v60,z0,tPen\WObj:=wPaper;
    MoveL Offs(pOrigin,264.45,312.49,0.00),v40,z0,tPen\WObj:=wPaper;
    MoveL Offs(pOrigin,263.60,312.27,0.00),v40,z0,tPen\WObj:=wPaper;
    MoveL Offs(pOrigin,263.60,312.27,0.00),v40,z0,tPen\WObj:=wPaper;
    MoveL Offs(pOrigin,259.14,311.21,0.00),v40,z0,tPen\WObj:=wPaper;
    MoveL Offs(pOrigin,259.14,311.21,0.00),v40,z0,tPen\WObj:=wPaper;
    MoveL Offs(pOrigin,259.77,313.12,0.00),v40,fine,tPen\WObj:=wPaper;
    MoveL Offs(pOrigin,259.77,313.12,6.00),v60,z5,tPen\WObj:=wPaper;
    MoveL Offs(pOrigin,258.29,312.27,6.00),vTravel,z5,tPen\WObj:=wPaper;
    MoveL Offs(pOrigin,258.29,312.27,0.00),v60,z0,tPen\WObj:=wPaper;
    MoveL Offs(pOrigin,258.71,312.70,0.00),v40,z0,tPen\WObj:=wPaper;
    MoveL Offs(pOrigin,258.29,312.27,0.00),v40,fine,tPen\WObj:=wPaper;
    MoveL Offs(pOrigin,258.29,312.27,6.00),v60,z5,tPen\WObj:=wPaper;
    MoveL Offs(pOrigin,256.59,310.79,6.00),vTravel,z5,tPen\WObj:=wPaper;
    MoveL Offs(pOrigin,256.59,310.79,0.00),v60,z0,tPen\WObj:=wPaper;
    MoveL Offs(pOrigin,257.01,311.42,0.00),v40,z0,tPen\WObj:=wPaper;
    MoveL Offs(pOrigin,256.59,310.79,0.00),v40,fine,tPen\WObj:=wPaper;
    MoveL Offs(pOrigin,256.59,310.79,6.00),v60,z5,tPen\WObj:=wPaper;
    MoveL Offs(pOrigin,255.52,313.55,6.00),vTravel,z5,tPen\WObj:=wPaper;
    MoveL Offs(pOrigin,255.52,313.55,0.00),v60,z0,tPen\WObj:=wPaper;
    MoveL Offs(pOrigin,255.95,313.98,0.00),v40,z0,tPen\WObj:=wPaper;
    MoveL Offs(pOrigin,255.52,313.55,0.00),v40,fine,tPen\WObj:=wPaper;
    MoveL Offs(pOrigin,255.52,313.55,6.00),v60,z5,tPen\WObj:=wPaper;
    MoveL Offs(pOrigin,253.19,313.98,6.00),vTravel,z5,tPen\WObj:=wPaper;
    MoveL Offs(pOrigin,253.19,313.98,0.00),v60,z0,tPen\WObj:=wPaper;
    MoveL Offs(pOrigin,253.82,314.61,0.00),v40,z0,tPen\WObj:=wPaper;
    MoveL Offs(pOrigin,253.19,313.98,0.00),v40,fine,tPen\WObj:=wPaper;
    MoveL Offs(pOrigin,253.19,313.98,6.00),v60,z5,tPen\WObj:=wPaper;
    MoveL Offs(pOrigin,252.55,312.49,6.00),vTravel,z5,tPen\WObj:=wPaper;
    MoveL Offs(pOrigin,252.55,312.49,0.00),v60,z0,tPen\WObj:=wPaper;
    MoveL Offs(pOrigin,252.98,313.55,0.00),v40,z0,tPen\WObj:=wPaper;
    MoveL Offs(pOrigin,254.82,315.67,0.00),v40,z0,tPen\WObj:=wPaper;
    MoveL Offs(pOrigin,255.31,318.01,0.00),v40,z0,tPen\WObj:=wPaper;
    MoveL Offs(pOrigin,256.16,318.44,0.00),v40,z0,tPen\WObj:=wPaper;
    MoveL Offs(pOrigin,256.66,320.14,0.00),v40,z0,tPen\WObj:=wPaper;
    MoveL Offs(pOrigin,257.65,320.99,0.00),v40,z0,tPen\WObj:=wPaper;
    MoveL Offs(pOrigin,258.71,321.20,0.00),v40,z0,tPen\WObj:=wPaper;
    MoveL Offs(pOrigin,259.35,321.84,0.00),v40,z0,tPen\WObj:=wPaper;
    MoveL Offs(pOrigin,258.71,321.20,0.00),v40,fine,tPen\WObj:=wPaper;
    MoveL Offs(pOrigin,258.71,321.20,6.00),v60,z5,tPen\WObj:=wPaper;
    MoveL Offs(pOrigin,252.12,319.08,6.00),vTravel,z5,tPen\WObj:=wPaper;
    MoveL Offs(pOrigin,252.12,319.08,0.00),v60,z0,tPen\WObj:=wPaper;
    MoveL Offs(pOrigin,249.79,318.65,0.00),v40,z0,tPen\WObj:=wPaper;
    MoveL Offs(pOrigin,248.94,319.08,0.00),v40,z0,tPen\WObj:=wPaper;
    MoveL Offs(pOrigin,247.45,318.86,0.00),v40,fine,tPen\WObj:=wPaper;
    MoveL Offs(pOrigin,247.45,318.86,6.00),v60,z5,tPen\WObj:=wPaper;
    MoveL Offs(pOrigin,246.60,321.20,6.00),vTravel,z5,tPen\WObj:=wPaper;
    MoveL Offs(pOrigin,246.60,321.20,0.00),v60,z0,tPen\WObj:=wPaper;
    MoveL Offs(pOrigin,247.02,321.41,0.00),v40,z0,tPen\WObj:=wPaper;
    MoveL Offs(pOrigin,246.60,321.20,0.00),v40,fine,tPen\WObj:=wPaper;
    MoveL Offs(pOrigin,246.60,321.20,6.00),v60,z5,tPen\WObj:=wPaper;
    MoveL Offs(pOrigin,244.69,319.92,6.00),vTravel,z5,tPen\WObj:=wPaper;
    MoveL Offs(pOrigin,244.69,319.92,0.00),v60,z0,tPen\WObj:=wPaper;
    MoveL Offs(pOrigin,245.54,320.70,0.00),v40,z0,tPen\WObj:=wPaper;
    MoveL Offs(pOrigin,247.24,321.41,0.00),v40,z0,tPen\WObj:=wPaper;
    MoveL Offs(pOrigin,248.73,323.47,0.00),v40,z0,tPen\WObj:=wPaper;
    MoveL Offs(pOrigin,250.43,324.17,0.00),v40,z0,tPen\WObj:=wPaper;
    MoveL Offs(pOrigin,252.27,326.16,0.00),v40,z0,tPen\WObj:=wPaper;
    MoveL Offs(pOrigin,252.55,329.06,0.00),v40,z0,tPen\WObj:=wPaper;
    MoveL Offs(pOrigin,251.77,331.19,0.00),v40,z0,tPen\WObj:=wPaper;
    MoveL Offs(pOrigin,250.85,331.61,0.00),v40,z0,tPen\WObj:=wPaper;
    MoveL Offs(pOrigin,250.85,331.61,0.00),v40,z0,tPen\WObj:=wPaper;
    MoveL Offs(pOrigin,250.43,332.67,0.00),v40,z0,tPen\WObj:=wPaper;
    MoveL Offs(pOrigin,249.15,333.52,0.00),v40,z0,tPen\WObj:=wPaper;
    MoveL Offs(pOrigin,249.15,333.95,0.00),v40,z0,tPen\WObj:=wPaper;
    MoveL Offs(pOrigin,247.45,334.23,0.00),v40,z0,tPen\WObj:=wPaper;
    MoveL Offs(pOrigin,246.39,335.23,0.00),v40,z0,tPen\WObj:=wPaper;
    MoveL Offs(pOrigin,247.02,334.59,0.00),v40,z0,tPen\WObj:=wPaper;
    MoveL Offs(pOrigin,246.81,335.01,0.00),v40,z0,tPen\WObj:=wPaper;
    MoveL Offs(pOrigin,247.02,334.59,0.00),v40,fine,tPen\WObj:=wPaper;
    MoveL Offs(pOrigin,247.02,334.59,6.00),v60,z5,tPen\WObj:=wPaper;
  ENDPROC

  PROC DrawPart73()
    MoveL Offs(pOrigin,247.66,336.29,6.00),vTravel,z5,tPen\WObj:=wPaper;
    MoveL Offs(pOrigin,247.66,336.29,0.00),v60,z0,tPen\WObj:=wPaper;
    MoveL Offs(pOrigin,248.09,336.08,0.00),v40,z0,tPen\WObj:=wPaper;
    MoveL Offs(pOrigin,247.66,336.29,0.00),v40,z0,tPen\WObj:=wPaper;
    MoveL Offs(pOrigin,247.24,336.50,0.00),v40,z0,tPen\WObj:=wPaper;
    MoveL Offs(pOrigin,248.65,335.65,0.00),v40,z0,tPen\WObj:=wPaper;
    MoveL Offs(pOrigin,249.15,334.59,0.00),v40,fine,tPen\WObj:=wPaper;
    MoveL Offs(pOrigin,249.15,334.59,6.00),v60,z5,tPen\WObj:=wPaper;
    MoveL Offs(pOrigin,250.64,334.38,6.00),vTravel,z5,tPen\WObj:=wPaper;
    MoveL Offs(pOrigin,250.64,334.38,0.00),v60,z0,tPen\WObj:=wPaper;
    MoveL Offs(pOrigin,250.85,333.95,0.00),v40,z0,tPen\WObj:=wPaper;
    MoveL Offs(pOrigin,250.64,334.38,0.00),v40,z0,tPen\WObj:=wPaper;
    MoveL Offs(pOrigin,251.27,333.74,0.00),v40,z0,tPen\WObj:=wPaper;
    MoveL Offs(pOrigin,251.49,333.31,0.00),v40,z0,tPen\WObj:=wPaper;
    MoveL Offs(pOrigin,251.27,333.74,0.00),v40,z0,tPen\WObj:=wPaper;
    MoveL Offs(pOrigin,251.91,333.10,0.00),v40,z0,tPen\WObj:=wPaper;
    MoveL Offs(pOrigin,252.12,332.67,0.00),v40,z0,tPen\WObj:=wPaper;
    MoveL Offs(pOrigin,251.91,333.10,0.00),v40,fine,tPen\WObj:=wPaper;
    MoveL Offs(pOrigin,251.91,333.10,6.00),v60,z5,tPen\WObj:=wPaper;
    MoveL Offs(pOrigin,252.34,334.80,6.00),vTravel,z5,tPen\WObj:=wPaper;
    MoveL Offs(pOrigin,252.34,334.80,0.00),v60,z0,tPen\WObj:=wPaper;
    MoveL Offs(pOrigin,254.60,332.46,0.00),v40,z0,tPen\WObj:=wPaper;
    MoveL Offs(pOrigin,255.31,330.76,0.00),v40,fine,tPen\WObj:=wPaper;
    MoveL Offs(pOrigin,255.31,330.76,6.00),v60,z5,tPen\WObj:=wPaper;
    MoveL Offs(pOrigin,250.85,331.61,6.00),vTravel,z5,tPen\WObj:=wPaper;
    MoveL Offs(pOrigin,250.85,331.61,0.00),v60,z0,tPen\WObj:=wPaper;
    MoveL Offs(pOrigin,251.06,328.64,0.00),v40,z0,tPen\WObj:=wPaper;
    MoveL Offs(pOrigin,250.43,326.09,0.00),v40,z0,tPen\WObj:=wPaper;
    MoveL Offs(pOrigin,250.85,325.02,0.00),v40,fine,tPen\WObj:=wPaper;
    MoveL Offs(pOrigin,250.85,325.02,6.00),v60,z5,tPen\WObj:=wPaper;
    MoveL Offs(pOrigin,246.39,323.96,6.00),vTravel,z5,tPen\WObj:=wPaper;
    MoveL Offs(pOrigin,246.39,323.96,0.00),v60,z0,tPen\WObj:=wPaper;
    MoveL Offs(pOrigin,247.66,327.58,0.00),v40,z0,tPen\WObj:=wPaper;
    MoveL Offs(pOrigin,247.66,330.55,0.00),v40,z0,tPen\WObj:=wPaper;
    MoveL Offs(pOrigin,246.67,333.10,0.00),v40,z0,tPen\WObj:=wPaper;
    MoveL Offs(pOrigin,245.96,333.52,0.00),v40,z0,tPen\WObj:=wPaper;
    MoveL Offs(pOrigin,245.11,333.52,0.00),v40,z0,tPen\WObj:=wPaper;
    MoveL Offs(pOrigin,245.11,333.52,0.00),v40,z0,tPen\WObj:=wPaper;
    MoveL Offs(pOrigin,244.05,335.01,0.00),v40,z0,tPen\WObj:=wPaper;
    MoveL Offs(pOrigin,244.05,335.65,0.00),v40,z0,tPen\WObj:=wPaper;
    MoveL Offs(pOrigin,243.20,336.08,0.00),v40,z0,tPen\WObj:=wPaper;
    MoveL Offs(pOrigin,242.99,335.65,0.00),v40,z0,tPen\WObj:=wPaper;
    MoveL Offs(pOrigin,241.50,335.65,0.00),v40,fine,tPen\WObj:=wPaper;
    MoveL Offs(pOrigin,241.50,335.65,6.00),v60,z5,tPen\WObj:=wPaper;
    MoveL Offs(pOrigin,242.14,334.59,6.00),vTravel,z5,tPen\WObj:=wPaper;
    MoveL Offs(pOrigin,242.14,334.59,0.00),v60,z0,tPen\WObj:=wPaper;
    MoveL Offs(pOrigin,242.35,334.16,0.00),v40,z0,tPen\WObj:=wPaper;
    MoveL Offs(pOrigin,242.14,334.59,0.00),v40,z0,tPen\WObj:=wPaper;
    MoveL Offs(pOrigin,242.77,333.95,0.00),v40,z0,tPen\WObj:=wPaper;
    MoveL Offs(pOrigin,242.99,333.52,0.00),v40,z0,tPen\WObj:=wPaper;
    MoveL Offs(pOrigin,242.77,333.95,0.00),v40,z0,tPen\WObj:=wPaper;
    MoveL Offs(pOrigin,243.41,333.10,0.00),v40,z0,tPen\WObj:=wPaper;
    MoveL Offs(pOrigin,243.62,332.67,0.00),v40,z0,tPen\WObj:=wPaper;
    MoveL Offs(pOrigin,243.41,333.10,0.00),v40,fine,tPen\WObj:=wPaper;
    MoveL Offs(pOrigin,243.41,333.10,6.00),v60,z5,tPen\WObj:=wPaper;
    MoveL Offs(pOrigin,245.54,335.65,6.00),vTravel,z5,tPen\WObj:=wPaper;
    MoveL Offs(pOrigin,245.54,335.65,0.00),v60,z0,tPen\WObj:=wPaper;
    MoveL Offs(pOrigin,245.82,335.51,0.00),v40,z0,tPen\WObj:=wPaper;
    MoveL Offs(pOrigin,244.90,336.00,0.00),v40,z0,tPen\WObj:=wPaper;
    MoveL Offs(pOrigin,243.84,335.79,0.00),v40,z0,tPen\WObj:=wPaper;
    MoveL Offs(pOrigin,242.77,336.85,0.00),v40,z0,tPen\WObj:=wPaper;
    MoveL Offs(pOrigin,240.01,337.99,0.00),v40,z0,tPen\WObj:=wPaper;
    MoveL Offs(pOrigin,237.25,338.62,0.00),v40,z0,tPen\WObj:=wPaper;
    MoveL Offs(pOrigin,236.40,338.41,0.00),v40,fine,tPen\WObj:=wPaper;
    MoveL Offs(pOrigin,236.40,338.41,6.00),v60,z5,tPen\WObj:=wPaper;
    MoveL Offs(pOrigin,244.05,338.41,6.00),vTravel,z5,tPen\WObj:=wPaper;
    MoveL Offs(pOrigin,244.05,338.41,0.00),v60,z0,tPen\WObj:=wPaper;
    MoveL Offs(pOrigin,245.32,338.62,0.00),v40,z0,tPen\WObj:=wPaper;
    MoveL Offs(pOrigin,245.32,338.62,0.00),v40,z0,tPen\WObj:=wPaper;
    MoveL Offs(pOrigin,245.32,338.84,0.00),v40,z0,tPen\WObj:=wPaper;
    MoveL Offs(pOrigin,246.39,338.62,0.00),v40,z0,tPen\WObj:=wPaper;
    MoveL Offs(pOrigin,246.39,337.99,0.00),v40,z0,tPen\WObj:=wPaper;
    MoveL Offs(pOrigin,246.39,338.41,0.00),v40,z0,tPen\WObj:=wPaper;
    MoveL Offs(pOrigin,247.02,338.62,0.00),v40,z0,tPen\WObj:=wPaper;
    MoveL Offs(pOrigin,247.45,337.99,0.00),v40,z0,tPen\WObj:=wPaper;
    MoveL Offs(pOrigin,247.45,337.99,0.00),v40,z0,tPen\WObj:=wPaper;
    MoveL Offs(pOrigin,250.21,337.77,0.00),v40,z0,tPen\WObj:=wPaper;
    MoveL Offs(pOrigin,252.55,337.14,0.00),v40,fine,tPen\WObj:=wPaper;
    MoveL Offs(pOrigin,252.55,337.14,6.00),v60,z5,tPen\WObj:=wPaper;
    MoveL Offs(pOrigin,252.98,335.86,6.00),vTravel,z5,tPen\WObj:=wPaper;
    MoveL Offs(pOrigin,252.98,335.86,0.00),v60,z0,tPen\WObj:=wPaper;
    MoveL Offs(pOrigin,252.62,336.92,0.00),v40,z0,tPen\WObj:=wPaper;
    MoveL Offs(pOrigin,254.04,337.14,0.00),v40,z0,tPen\WObj:=wPaper;
    MoveL Offs(pOrigin,254.04,337.14,0.00),v40,z0,tPen\WObj:=wPaper;
    MoveL Offs(pOrigin,254.89,337.63,0.00),v40,z0,tPen\WObj:=wPaper;
    MoveL Offs(pOrigin,257.65,336.29,0.00),v40,fine,tPen\WObj:=wPaper;
    MoveL Offs(pOrigin,257.65,336.29,6.00),v60,z5,tPen\WObj:=wPaper;
    MoveL Offs(pOrigin,254.68,336.08,6.00),vTravel,z5,tPen\WObj:=wPaper;
    MoveL Offs(pOrigin,254.68,336.08,0.00),v60,z0,tPen\WObj:=wPaper;
    MoveL Offs(pOrigin,255.52,335.65,0.00),v40,z0,tPen\WObj:=wPaper;
    MoveL Offs(pOrigin,255.95,334.45,0.00),v40,z0,tPen\WObj:=wPaper;
    MoveL Offs(pOrigin,255.10,334.52,0.00),v40,z0,tPen\WObj:=wPaper;
    MoveL Offs(pOrigin,254.25,335.44,0.00),v40,z0,tPen\WObj:=wPaper;
    MoveL Offs(pOrigin,254.25,335.44,0.00),v40,z0,tPen\WObj:=wPaper;
    MoveL Offs(pOrigin,253.61,335.44,0.00),v40,z0,tPen\WObj:=wPaper;
    MoveL Offs(pOrigin,253.40,335.86,0.00),v40,z0,tPen\WObj:=wPaper;
    MoveL Offs(pOrigin,253.61,335.65,0.00),v40,z0,tPen\WObj:=wPaper;
    MoveL Offs(pOrigin,254.68,336.08,0.00),v40,z0,tPen\WObj:=wPaper;
    MoveL Offs(pOrigin,254.04,337.14,0.00),v40,fine,tPen\WObj:=wPaper;
    MoveL Offs(pOrigin,254.04,337.14,6.00),v60,z5,tPen\WObj:=wPaper;
    MoveL Offs(pOrigin,247.45,337.99,6.00),vTravel,z5,tPen\WObj:=wPaper;
    MoveL Offs(pOrigin,247.45,337.99,0.00),v60,z0,tPen\WObj:=wPaper;
    MoveL Offs(pOrigin,247.45,337.77,0.00),v40,z0,tPen\WObj:=wPaper;
    MoveL Offs(pOrigin,246.39,337.99,0.00),v40,z0,tPen\WObj:=wPaper;
    MoveL Offs(pOrigin,246.39,337.99,0.00),v40,z0,tPen\WObj:=wPaper;
    MoveL Offs(pOrigin,245.75,337.99,0.00),v40,z0,tPen\WObj:=wPaper;
    MoveL Offs(pOrigin,245.32,338.62,0.00),v40,fine,tPen\WObj:=wPaper;
    MoveL Offs(pOrigin,245.32,338.62,6.00),v60,z5,tPen\WObj:=wPaper;
    MoveL Offs(pOrigin,244.05,338.41,6.00),vTravel,z5,tPen\WObj:=wPaper;
    MoveL Offs(pOrigin,244.05,338.41,0.00),v60,z0,tPen\WObj:=wPaper;
    MoveL Offs(pOrigin,244.26,337.77,0.00),v40,z0,tPen\WObj:=wPaper;
    MoveL Offs(pOrigin,246.60,336.71,0.00),v40,fine,tPen\WObj:=wPaper;
    MoveL Offs(pOrigin,246.60,336.71,6.00),v60,z5,tPen\WObj:=wPaper;
    MoveL Offs(pOrigin,238.10,321.84,6.00),vTravel,z5,tPen\WObj:=wPaper;
    MoveL Offs(pOrigin,238.10,321.84,0.00),v60,z0,tPen\WObj:=wPaper;
    MoveL Offs(pOrigin,237.04,320.77,0.00),v40,fine,tPen\WObj:=wPaper;
    MoveL Offs(pOrigin,237.04,320.77,6.00),v60,z5,tPen\WObj:=wPaper;
    MoveL Offs(pOrigin,240.44,320.14,6.00),vTravel,z5,tPen\WObj:=wPaper;
    MoveL Offs(pOrigin,240.44,320.14,0.00),v60,z0,tPen\WObj:=wPaper;
    MoveL Offs(pOrigin,241.29,320.99,0.00),v40,z0,tPen\WObj:=wPaper;
  ENDPROC

  PROC DrawPart74()
    MoveL Offs(pOrigin,240.44,320.14,0.00),v40,fine,tPen\WObj:=wPaper;
    MoveL Offs(pOrigin,240.44,320.14,6.00),v60,z5,tPen\WObj:=wPaper;
    MoveL Offs(pOrigin,238.74,317.59,6.00),vTravel,z5,tPen\WObj:=wPaper;
    MoveL Offs(pOrigin,238.74,317.59,0.00),v60,z0,tPen\WObj:=wPaper;
    MoveL Offs(pOrigin,238.31,313.34,0.00),v40,z0,tPen\WObj:=wPaper;
    MoveL Offs(pOrigin,238.67,312.06,0.00),v40,z0,tPen\WObj:=wPaper;
    MoveL Offs(pOrigin,239.59,311.42,0.00),v40,fine,tPen\WObj:=wPaper;
    MoveL Offs(pOrigin,239.59,311.42,6.00),v60,z5,tPen\WObj:=wPaper;
    MoveL Offs(pOrigin,238.74,310.15,6.00),vTravel,z5,tPen\WObj:=wPaper;
    MoveL Offs(pOrigin,238.74,310.15,0.00),v60,z0,tPen\WObj:=wPaper;
    MoveL Offs(pOrigin,238.17,310.36,0.00),v40,z0,tPen\WObj:=wPaper;
    MoveL Offs(pOrigin,237.25,312.06,0.00),v40,z0,tPen\WObj:=wPaper;
    MoveL Offs(pOrigin,237.25,312.06,0.00),v40,z0,tPen\WObj:=wPaper;
    MoveL Offs(pOrigin,236.68,312.49,0.00),v40,z0,tPen\WObj:=wPaper;
    MoveL Offs(pOrigin,236.33,314.19,0.00),v40,z0,tPen\WObj:=wPaper;
    MoveL Offs(pOrigin,235.98,314.40,0.00),v40,fine,tPen\WObj:=wPaper;
    MoveL Offs(pOrigin,235.98,314.40,6.00),v60,z5,tPen\WObj:=wPaper;
    MoveL Offs(pOrigin,237.25,312.06,6.00),vTravel,z5,tPen\WObj:=wPaper;
    MoveL Offs(pOrigin,237.25,312.06,0.00),v60,z0,tPen\WObj:=wPaper;
    MoveL Offs(pOrigin,237.46,312.49,0.00),v40,z0,tPen\WObj:=wPaper;
    MoveL Offs(pOrigin,237.25,314.83,0.00),v40,z0,tPen\WObj:=wPaper;
    MoveL Offs(pOrigin,237.68,316.95,0.00),v40,fine,tPen\WObj:=wPaper;
    MoveL Offs(pOrigin,237.68,316.95,6.00),v60,z5,tPen\WObj:=wPaper;
    MoveL Offs(pOrigin,240.01,316.10,6.00),vTravel,z5,tPen\WObj:=wPaper;
    MoveL Offs(pOrigin,240.01,316.10,0.00),v60,z0,tPen\WObj:=wPaper;
    MoveL Offs(pOrigin,240.23,316.52,0.00),v40,z0,tPen\WObj:=wPaper;
    MoveL Offs(pOrigin,240.01,316.10,0.00),v40,fine,tPen\WObj:=wPaper;
    MoveL Offs(pOrigin,240.01,316.10,6.00),v60,z5,tPen\WObj:=wPaper;
    MoveL Offs(pOrigin,206.23,260.85,6.00),vTravel,z5,tPen\WObj:=wPaper;
    MoveL Offs(pOrigin,206.23,260.85,0.00),v60,z0,tPen\WObj:=wPaper;
    MoveL Offs(pOrigin,206.01,261.27,0.00),v40,z0,tPen\WObj:=wPaper;
    MoveL Offs(pOrigin,206.23,260.85,0.00),v40,fine,tPen\WObj:=wPaper;
    MoveL Offs(pOrigin,206.23,260.85,6.00),v60,z5,tPen\WObj:=wPaper;
    MoveL Offs(pOrigin,207.93,258.94,6.00),vTravel,z5,tPen\WObj:=wPaper;
    MoveL Offs(pOrigin,207.93,258.94,0.00),v60,z0,tPen\WObj:=wPaper;
    MoveL Offs(pOrigin,207.07,258.73,0.00),v40,z0,tPen\WObj:=wPaper;
    MoveL Offs(pOrigin,207.29,257.88,0.00),v40,z0,tPen\WObj:=wPaper;
    MoveL Offs(pOrigin,207.07,257.88,0.00),v40,z0,tPen\WObj:=wPaper;
    MoveL Offs(pOrigin,207.71,257.66,0.00),v40,z0,tPen\WObj:=wPaper;
    MoveL Offs(pOrigin,208.14,258.09,0.00),v40,z0,tPen\WObj:=wPaper;
    MoveL Offs(pOrigin,207.71,257.66,0.00),v40,fine,tPen\WObj:=wPaper;
    MoveL Offs(pOrigin,207.71,257.66,6.00),v60,z5,tPen\WObj:=wPaper;
    MoveL Offs(pOrigin,201.98,261.91,6.00),vTravel,z5,tPen\WObj:=wPaper;
    MoveL Offs(pOrigin,201.98,261.91,0.00),v60,z0,tPen\WObj:=wPaper;
    MoveL Offs(pOrigin,200.70,263.19,0.00),v40,z0,tPen\WObj:=wPaper;
    MoveL Offs(pOrigin,199.00,263.12,0.00),v40,z0,tPen\WObj:=wPaper;
    MoveL Offs(pOrigin,197.73,262.12,0.00),v40,z0,tPen\WObj:=wPaper;
    MoveL Offs(pOrigin,196.80,260.42,0.00),v40,z0,tPen\WObj:=wPaper;
    MoveL Offs(pOrigin,196.24,258.30,0.00),v40,z0,tPen\WObj:=wPaper;
    MoveL Offs(pOrigin,196.24,254.48,0.00),v40,z0,tPen\WObj:=wPaper;
    MoveL Offs(pOrigin,196.80,252.14,0.00),v40,z0,tPen\WObj:=wPaper;
    MoveL Offs(pOrigin,200.98,244.91,0.00),v40,z0,tPen\WObj:=wPaper;
    MoveL Offs(pOrigin,202.47,240.66,0.00),v40,z0,tPen\WObj:=wPaper;
    MoveL Offs(pOrigin,203.46,236.41,0.00),v40,z0,tPen\WObj:=wPaper;
    MoveL Offs(pOrigin,203.68,232.38,0.00),v40,z0,tPen\WObj:=wPaper;
    MoveL Offs(pOrigin,204.03,231.10,0.00),v40,z0,tPen\WObj:=wPaper;
    MoveL Offs(pOrigin,204.95,229.40,0.00),v40,z0,tPen\WObj:=wPaper;
    MoveL Offs(pOrigin,206.44,228.34,0.00),v40,z0,tPen\WObj:=wPaper;
    MoveL Offs(pOrigin,207.29,228.34,0.00),v40,z0,tPen\WObj:=wPaper;
    MoveL Offs(pOrigin,207.71,228.76,0.00),v40,z0,tPen\WObj:=wPaper;
    MoveL Offs(pOrigin,207.29,232.38,0.00),v40,z0,tPen\WObj:=wPaper;
    MoveL Offs(pOrigin,207.29,232.38,0.00),v40,z0,tPen\WObj:=wPaper;
    MoveL Offs(pOrigin,207.07,233.44,0.00),v40,z0,tPen\WObj:=wPaper;
    MoveL Offs(pOrigin,207.29,233.65,0.00),v40,fine,tPen\WObj:=wPaper;
    MoveL Offs(pOrigin,207.29,233.65,6.00),v60,z5,tPen\WObj:=wPaper;
    MoveL Offs(pOrigin,205.38,228.76,6.00),vTravel,z5,tPen\WObj:=wPaper;
    MoveL Offs(pOrigin,205.38,228.76,0.00),v60,z0,tPen\WObj:=wPaper;
    MoveL Offs(pOrigin,204.74,229.40,0.00),v40,z0,tPen\WObj:=wPaper;
    MoveL Offs(pOrigin,205.38,228.76,0.00),v40,fine,tPen\WObj:=wPaper;
    MoveL Offs(pOrigin,205.38,228.76,6.00),v60,z5,tPen\WObj:=wPaper;
    MoveL Offs(pOrigin,204.31,227.91,6.00),vTravel,z5,tPen\WObj:=wPaper;
    MoveL Offs(pOrigin,204.31,227.91,0.00),v60,z0,tPen\WObj:=wPaper;
    MoveL Offs(pOrigin,203.89,228.34,0.00),v40,z0,tPen\WObj:=wPaper;
    MoveL Offs(pOrigin,204.31,227.91,0.00),v40,z0,tPen\WObj:=wPaper;
    MoveL Offs(pOrigin,203.68,228.55,0.00),v40,z0,tPen\WObj:=wPaper;
    MoveL Offs(pOrigin,203.25,229.19,0.00),v40,z0,tPen\WObj:=wPaper;
    MoveL Offs(pOrigin,203.68,228.55,0.00),v40,fine,tPen\WObj:=wPaper;
    MoveL Offs(pOrigin,203.68,228.55,6.00),v60,z5,tPen\WObj:=wPaper;
    MoveL Offs(pOrigin,210.48,224.30,6.00),vTravel,z5,tPen\WObj:=wPaper;
    MoveL Offs(pOrigin,210.48,224.30,0.00),v60,z0,tPen\WObj:=wPaper;
    MoveL Offs(pOrigin,210.26,224.73,0.00),v40,z0,tPen\WObj:=wPaper;
    MoveL Offs(pOrigin,210.48,224.30,0.00),v40,fine,tPen\WObj:=wPaper;
    MoveL Offs(pOrigin,210.48,224.30,6.00),v60,z5,tPen\WObj:=wPaper;
    MoveL Offs(pOrigin,211.11,223.02,6.00),vTravel,z5,tPen\WObj:=wPaper;
    MoveL Offs(pOrigin,211.11,223.02,0.00),v60,z0,tPen\WObj:=wPaper;
    MoveL Offs(pOrigin,210.90,223.45,0.00),v40,z0,tPen\WObj:=wPaper;
    MoveL Offs(pOrigin,211.11,223.02,0.00),v40,z0,tPen\WObj:=wPaper;
    MoveL Offs(pOrigin,211.54,222.18,0.00),v40,z0,tPen\WObj:=wPaper;
    MoveL Offs(pOrigin,211.32,222.60,0.00),v40,z0,tPen\WObj:=wPaper;
    MoveL Offs(pOrigin,211.54,222.18,0.00),v40,fine,tPen\WObj:=wPaper;
    MoveL Offs(pOrigin,211.54,222.18,6.00),v60,z5,tPen\WObj:=wPaper;
    MoveL Offs(pOrigin,209.84,222.39,6.00),vTravel,z5,tPen\WObj:=wPaper;
    MoveL Offs(pOrigin,209.84,222.39,0.00),v60,z0,tPen\WObj:=wPaper;
    MoveL Offs(pOrigin,209.62,222.81,0.00),v40,z0,tPen\WObj:=wPaper;
    MoveL Offs(pOrigin,209.84,222.39,0.00),v40,fine,tPen\WObj:=wPaper;
    MoveL Offs(pOrigin,209.84,222.39,6.00),v60,z5,tPen\WObj:=wPaper;
    MoveL Offs(pOrigin,212.81,220.05,6.00),vTravel,z5,tPen\WObj:=wPaper;
    MoveL Offs(pOrigin,212.81,220.05,0.00),v60,z0,tPen\WObj:=wPaper;
    MoveL Offs(pOrigin,212.39,220.69,0.00),v40,z0,tPen\WObj:=wPaper;
    MoveL Offs(pOrigin,212.81,220.05,0.00),v40,fine,tPen\WObj:=wPaper;
    MoveL Offs(pOrigin,212.81,220.05,6.00),v60,z5,tPen\WObj:=wPaper;
    MoveL Offs(pOrigin,212.39,218.35,6.00),vTravel,z5,tPen\WObj:=wPaper;
    MoveL Offs(pOrigin,212.39,218.35,0.00),v60,z0,tPen\WObj:=wPaper;
    MoveL Offs(pOrigin,211.96,218.77,0.00),v40,z0,tPen\WObj:=wPaper;
    MoveL Offs(pOrigin,212.39,218.35,0.00),v40,fine,tPen\WObj:=wPaper;
    MoveL Offs(pOrigin,212.39,218.35,6.00),v60,z5,tPen\WObj:=wPaper;
    MoveL Offs(pOrigin,213.66,216.86,6.00),vTravel,z5,tPen\WObj:=wPaper;
    MoveL Offs(pOrigin,213.66,216.86,0.00),v60,z0,tPen\WObj:=wPaper;
    MoveL Offs(pOrigin,212.60,217.93,0.00),v40,z0,tPen\WObj:=wPaper;
    MoveL Offs(pOrigin,213.66,216.86,0.00),v40,fine,tPen\WObj:=wPaper;
    MoveL Offs(pOrigin,213.66,216.86,6.00),v60,z5,tPen\WObj:=wPaper;
    MoveL Offs(pOrigin,214.73,217.71,6.00),vTravel,z5,tPen\WObj:=wPaper;
    MoveL Offs(pOrigin,214.73,217.71,0.00),v60,z0,tPen\WObj:=wPaper;
    MoveL Offs(pOrigin,213.88,218.56,0.00),v40,z0,tPen\WObj:=wPaper;
    MoveL Offs(pOrigin,214.73,217.71,0.00),v40,fine,tPen\WObj:=wPaper;
    MoveL Offs(pOrigin,214.73,217.71,6.00),v60,z5,tPen\WObj:=wPaper;
    MoveL Offs(pOrigin,215.15,215.16,6.00),vTravel,z5,tPen\WObj:=wPaper;
    MoveL Offs(pOrigin,215.15,215.16,0.00),v60,z0,tPen\WObj:=wPaper;
    MoveL Offs(pOrigin,213.88,216.44,0.00),v40,z0,tPen\WObj:=wPaper;
    MoveL Offs(pOrigin,215.15,215.16,0.00),v40,fine,tPen\WObj:=wPaper;
  ENDPROC

  PROC DrawPart75()
    MoveL Offs(pOrigin,215.15,215.16,6.00),v60,z5,tPen\WObj:=wPaper;
    MoveL Offs(pOrigin,216.85,215.38,6.00),vTravel,z5,tPen\WObj:=wPaper;
    MoveL Offs(pOrigin,216.85,215.38,0.00),v60,z0,tPen\WObj:=wPaper;
    MoveL Offs(pOrigin,214.94,217.29,0.00),v40,z0,tPen\WObj:=wPaper;
    MoveL Offs(pOrigin,216.85,215.38,0.00),v40,fine,tPen\WObj:=wPaper;
    MoveL Offs(pOrigin,216.85,215.38,6.00),v60,z5,tPen\WObj:=wPaper;
    MoveL Offs(pOrigin,218.34,212.19,6.00),vTravel,z5,tPen\WObj:=wPaper;
    MoveL Offs(pOrigin,218.34,212.19,0.00),v60,z0,tPen\WObj:=wPaper;
    MoveL Offs(pOrigin,217.91,212.33,0.00),v40,z0,tPen\WObj:=wPaper;
    MoveL Offs(pOrigin,217.27,211.98,0.00),v40,z0,tPen\WObj:=wPaper;
    MoveL Offs(pOrigin,213.02,207.51,0.00),v40,z0,tPen\WObj:=wPaper;
    MoveL Offs(pOrigin,198.29,190.09,0.00),v40,z0,tPen\WObj:=wPaper;
    MoveL Offs(pOrigin,198.57,189.52,0.00),v40,z0,tPen\WObj:=wPaper;
    MoveL Offs(pOrigin,208.56,186.05,0.00),v40,z0,tPen\WObj:=wPaper;
    MoveL Offs(pOrigin,209.62,186.19,0.00),v40,z0,tPen\WObj:=wPaper;
    MoveL Offs(pOrigin,212.60,188.18,0.00),v40,z0,tPen\WObj:=wPaper;
    MoveL Offs(pOrigin,212.60,188.18,0.00),v40,z0,tPen\WObj:=wPaper;
    MoveL Offs(pOrigin,213.88,188.81,0.00),v40,fine,tPen\WObj:=wPaper;
    MoveL Offs(pOrigin,213.88,188.81,6.00),v60,z5,tPen\WObj:=wPaper;
    MoveL Offs(pOrigin,210.05,186.69,6.00),vTravel,z5,tPen\WObj:=wPaper;
    MoveL Offs(pOrigin,210.05,186.69,0.00),v60,z0,tPen\WObj:=wPaper;
    MoveL Offs(pOrigin,210.69,187.11,0.00),v40,z0,tPen\WObj:=wPaper;
    MoveL Offs(pOrigin,210.05,186.69,0.00),v40,z0,tPen\WObj:=wPaper;
    MoveL Offs(pOrigin,209.41,186.26,0.00),v40,z0,tPen\WObj:=wPaper;
    MoveL Offs(pOrigin,209.84,186.48,0.00),v40,z0,tPen\WObj:=wPaper;
    MoveL Offs(pOrigin,209.41,186.26,0.00),v40,fine,tPen\WObj:=wPaper;
    MoveL Offs(pOrigin,209.41,186.26,6.00),v60,z5,tPen\WObj:=wPaper;
    MoveL Offs(pOrigin,208.99,184.77,6.00),vTravel,z5,tPen\WObj:=wPaper;
    MoveL Offs(pOrigin,208.99,184.77,0.00),v60,z0,tPen\WObj:=wPaper;
    MoveL Offs(pOrigin,209.41,184.99,0.00),v40,z0,tPen\WObj:=wPaper;
    MoveL Offs(pOrigin,208.99,184.77,0.00),v40,z0,tPen\WObj:=wPaper;
    MoveL Offs(pOrigin,208.35,184.35,0.00),v40,z0,tPen\WObj:=wPaper;
    MoveL Offs(pOrigin,208.77,184.56,0.00),v40,z0,tPen\WObj:=wPaper;
    MoveL Offs(pOrigin,208.35,184.35,0.00),v40,z0,tPen\WObj:=wPaper;
    MoveL Offs(pOrigin,207.50,183.93,0.00),v40,z0,tPen\WObj:=wPaper;
    MoveL Offs(pOrigin,207.93,184.14,0.00),v40,z0,tPen\WObj:=wPaper;
    MoveL Offs(pOrigin,207.50,183.93,0.00),v40,fine,tPen\WObj:=wPaper;
    MoveL Offs(pOrigin,207.50,183.93,6.00),v60,z5,tPen\WObj:=wPaper;
    MoveL Offs(pOrigin,205.59,182.86,6.00),vTravel,z5,tPen\WObj:=wPaper;
    MoveL Offs(pOrigin,205.59,182.86,0.00),v60,z0,tPen\WObj:=wPaper;
    MoveL Offs(pOrigin,206.01,183.07,0.00),v40,z0,tPen\WObj:=wPaper;
    MoveL Offs(pOrigin,205.59,182.86,0.00),v40,fine,tPen\WObj:=wPaper;
    MoveL Offs(pOrigin,205.59,182.86,6.00),v60,z5,tPen\WObj:=wPaper;
    MoveL Offs(pOrigin,204.52,182.23,6.00),vTravel,z5,tPen\WObj:=wPaper;
    MoveL Offs(pOrigin,204.52,182.23,0.00),v60,z0,tPen\WObj:=wPaper;
    MoveL Offs(pOrigin,204.95,182.44,0.00),v40,z0,tPen\WObj:=wPaper;
    MoveL Offs(pOrigin,204.52,182.23,0.00),v40,z0,tPen\WObj:=wPaper;
    MoveL Offs(pOrigin,203.68,181.80,0.00),v40,z0,tPen\WObj:=wPaper;
    MoveL Offs(pOrigin,204.10,182.01,0.00),v40,z0,tPen\WObj:=wPaper;
    MoveL Offs(pOrigin,203.68,181.80,0.00),v40,z0,tPen\WObj:=wPaper;
    MoveL Offs(pOrigin,202.82,181.38,0.00),v40,z0,tPen\WObj:=wPaper;
    MoveL Offs(pOrigin,203.25,181.59,0.00),v40,z0,tPen\WObj:=wPaper;
    MoveL Offs(pOrigin,202.82,181.38,0.00),v40,z0,tPen\WObj:=wPaper;
    MoveL Offs(pOrigin,201.98,180.95,0.00),v40,z0,tPen\WObj:=wPaper;
    MoveL Offs(pOrigin,202.40,181.16,0.00),v40,z0,tPen\WObj:=wPaper;
    MoveL Offs(pOrigin,201.98,180.95,0.00),v40,fine,tPen\WObj:=wPaper;
    MoveL Offs(pOrigin,201.98,180.95,6.00),v60,z5,tPen\WObj:=wPaper;
    MoveL Offs(pOrigin,200.91,180.31,6.00),vTravel,z5,tPen\WObj:=wPaper;
    MoveL Offs(pOrigin,200.91,180.31,0.00),v60,z0,tPen\WObj:=wPaper;
    MoveL Offs(pOrigin,201.34,180.52,0.00),v40,z0,tPen\WObj:=wPaper;
    MoveL Offs(pOrigin,200.91,180.31,0.00),v40,fine,tPen\WObj:=wPaper;
    MoveL Offs(pOrigin,200.91,180.31,6.00),v60,z5,tPen\WObj:=wPaper;
    MoveL Offs(pOrigin,199.64,179.68,6.00),vTravel,z5,tPen\WObj:=wPaper;
    MoveL Offs(pOrigin,199.64,179.68,0.00),v60,z0,tPen\WObj:=wPaper;
    MoveL Offs(pOrigin,200.06,179.89,0.00),v40,z0,tPen\WObj:=wPaper;
    MoveL Offs(pOrigin,199.64,179.68,0.00),v40,z0,tPen\WObj:=wPaper;
    MoveL Offs(pOrigin,198.79,179.25,0.00),v40,z0,tPen\WObj:=wPaper;
    MoveL Offs(pOrigin,199.21,179.46,0.00),v40,z0,tPen\WObj:=wPaper;
    MoveL Offs(pOrigin,198.79,179.25,0.00),v40,z0,tPen\WObj:=wPaper;
    MoveL Offs(pOrigin,197.94,178.82,0.00),v40,z0,tPen\WObj:=wPaper;
    MoveL Offs(pOrigin,198.36,179.04,0.00),v40,z0,tPen\WObj:=wPaper;
    MoveL Offs(pOrigin,197.94,178.82,0.00),v40,fine,tPen\WObj:=wPaper;
    MoveL Offs(pOrigin,197.94,178.82,6.00),v60,z5,tPen\WObj:=wPaper;
    MoveL Offs(pOrigin,197.30,179.89,6.00),vTravel,z5,tPen\WObj:=wPaper;
    MoveL Offs(pOrigin,197.30,179.89,0.00),v60,z0,tPen\WObj:=wPaper;
    MoveL Offs(pOrigin,197.73,180.10,0.00),v40,z0,tPen\WObj:=wPaper;
    MoveL Offs(pOrigin,197.30,179.89,0.00),v40,z0,tPen\WObj:=wPaper;
    MoveL Offs(pOrigin,198.15,180.31,0.00),v40,z0,tPen\WObj:=wPaper;
    MoveL Offs(pOrigin,198.79,180.74,0.00),v40,z0,tPen\WObj:=wPaper;
    MoveL Offs(pOrigin,198.15,180.31,0.00),v40,fine,tPen\WObj:=wPaper;
    MoveL Offs(pOrigin,198.15,180.31,6.00),v60,z5,tPen\WObj:=wPaper;
    MoveL Offs(pOrigin,199.64,181.16,6.00),vTravel,z5,tPen\WObj:=wPaper;
    MoveL Offs(pOrigin,199.64,181.16,0.00),v60,z0,tPen\WObj:=wPaper;
    MoveL Offs(pOrigin,200.06,181.38,0.00),v40,z0,tPen\WObj:=wPaper;
    MoveL Offs(pOrigin,199.64,181.16,0.00),v40,fine,tPen\WObj:=wPaper;
    MoveL Offs(pOrigin,199.64,181.16,6.00),v60,z5,tPen\WObj:=wPaper;
    MoveL Offs(pOrigin,200.91,181.80,6.00),vTravel,z5,tPen\WObj:=wPaper;
    MoveL Offs(pOrigin,200.91,181.80,0.00),v60,z0,tPen\WObj:=wPaper;
    MoveL Offs(pOrigin,201.34,182.01,0.00),v40,z0,tPen\WObj:=wPaper;
    MoveL Offs(pOrigin,200.91,181.80,0.00),v40,fine,tPen\WObj:=wPaper;
    MoveL Offs(pOrigin,200.91,181.80,6.00),v60,z5,tPen\WObj:=wPaper;
    MoveL Offs(pOrigin,202.19,182.44,6.00),vTravel,z5,tPen\WObj:=wPaper;
    MoveL Offs(pOrigin,202.19,182.44,0.00),v60,z0,tPen\WObj:=wPaper;
    MoveL Offs(pOrigin,202.82,182.86,0.00),v40,z0,tPen\WObj:=wPaper;
    MoveL Offs(pOrigin,202.19,182.44,0.00),v40,fine,tPen\WObj:=wPaper;
    MoveL Offs(pOrigin,202.19,182.44,6.00),v60,z5,tPen\WObj:=wPaper;
    MoveL Offs(pOrigin,203.68,183.29,6.00),vTravel,z5,tPen\WObj:=wPaper;
    MoveL Offs(pOrigin,203.68,183.29,0.00),v60,z0,tPen\WObj:=wPaper;
    MoveL Offs(pOrigin,204.10,183.50,0.00),v40,z0,tPen\WObj:=wPaper;
    MoveL Offs(pOrigin,203.68,183.29,0.00),v40,z0,tPen\WObj:=wPaper;
    MoveL Offs(pOrigin,204.52,183.71,0.00),v40,z0,tPen\WObj:=wPaper;
    MoveL Offs(pOrigin,204.95,183.93,0.00),v40,z0,tPen\WObj:=wPaper;
    MoveL Offs(pOrigin,204.52,183.71,0.00),v40,fine,tPen\WObj:=wPaper;
    MoveL Offs(pOrigin,204.52,183.71,6.00),v60,z5,tPen\WObj:=wPaper;
    MoveL Offs(pOrigin,199.85,191.79,6.00),vTravel,z5,tPen\WObj:=wPaper;
    MoveL Offs(pOrigin,199.85,191.79,0.00),v60,z0,tPen\WObj:=wPaper;
    MoveL Offs(pOrigin,200.06,192.21,0.00),v40,z0,tPen\WObj:=wPaper;
    MoveL Offs(pOrigin,199.85,191.79,0.00),v40,z0,tPen\WObj:=wPaper;
    MoveL Offs(pOrigin,200.27,192.43,0.00),v40,z0,tPen\WObj:=wPaper;
    MoveL Offs(pOrigin,200.70,192.85,0.00),v40,z0,tPen\WObj:=wPaper;
    MoveL Offs(pOrigin,200.27,192.43,0.00),v40,fine,tPen\WObj:=wPaper;
    MoveL Offs(pOrigin,200.27,192.43,6.00),v60,z5,tPen\WObj:=wPaper;
    MoveL Offs(pOrigin,201.34,193.49,6.00),vTravel,z5,tPen\WObj:=wPaper;
    MoveL Offs(pOrigin,201.34,193.49,0.00),v60,z0,tPen\WObj:=wPaper;
    MoveL Offs(pOrigin,202.40,194.76,0.00),v40,z0,tPen\WObj:=wPaper;
    MoveL Offs(pOrigin,201.34,193.49,0.00),v40,fine,tPen\WObj:=wPaper;
    MoveL Offs(pOrigin,201.34,193.49,6.00),v60,z5,tPen\WObj:=wPaper;
    MoveL Offs(pOrigin,200.27,194.76,6.00),vTravel,z5,tPen\WObj:=wPaper;
    MoveL Offs(pOrigin,200.27,194.76,0.00),v60,z0,tPen\WObj:=wPaper;
    MoveL Offs(pOrigin,200.91,195.40,0.00),v40,z0,tPen\WObj:=wPaper;
  ENDPROC

  PROC DrawPart76()
    MoveL Offs(pOrigin,200.27,194.76,0.00),v40,fine,tPen\WObj:=wPaper;
    MoveL Offs(pOrigin,200.27,194.76,6.00),v60,z5,tPen\WObj:=wPaper;
    MoveL Offs(pOrigin,199.00,193.27,6.00),vTravel,z5,tPen\WObj:=wPaper;
    MoveL Offs(pOrigin,199.00,193.27,0.00),v60,z0,tPen\WObj:=wPaper;
    MoveL Offs(pOrigin,199.64,193.91,0.00),v40,z0,tPen\WObj:=wPaper;
    MoveL Offs(pOrigin,199.00,193.27,0.00),v40,fine,tPen\WObj:=wPaper;
    MoveL Offs(pOrigin,199.00,193.27,6.00),v60,z5,tPen\WObj:=wPaper;
    MoveL Offs(pOrigin,197.94,192.00,6.00),vTravel,z5,tPen\WObj:=wPaper;
    MoveL Offs(pOrigin,197.94,192.00,0.00),v60,z0,tPen\WObj:=wPaper;
    MoveL Offs(pOrigin,198.79,192.85,0.00),v40,z0,tPen\WObj:=wPaper;
    MoveL Offs(pOrigin,197.94,192.00,0.00),v40,fine,tPen\WObj:=wPaper;
    MoveL Offs(pOrigin,197.94,192.00,6.00),v60,z5,tPen\WObj:=wPaper;
    MoveL Offs(pOrigin,196.88,190.73,6.00),vTravel,z5,tPen\WObj:=wPaper;
    MoveL Offs(pOrigin,196.88,190.73,0.00),v60,z0,tPen\WObj:=wPaper;
    MoveL Offs(pOrigin,197.51,191.36,0.00),v40,z0,tPen\WObj:=wPaper;
    MoveL Offs(pOrigin,196.88,190.73,0.00),v40,fine,tPen\WObj:=wPaper;
    MoveL Offs(pOrigin,196.88,190.73,6.00),v60,z5,tPen\WObj:=wPaper;
    MoveL Offs(pOrigin,201.55,196.25,6.00),vTravel,z5,tPen\WObj:=wPaper;
    MoveL Offs(pOrigin,201.55,196.25,0.00),v60,z0,tPen\WObj:=wPaper;
    MoveL Offs(pOrigin,201.98,196.68,0.00),v40,z0,tPen\WObj:=wPaper;
    MoveL Offs(pOrigin,201.55,196.25,0.00),v40,z0,tPen\WObj:=wPaper;
    MoveL Offs(pOrigin,202.19,197.10,0.00),v40,z0,tPen\WObj:=wPaper;
    MoveL Offs(pOrigin,203.25,198.16,0.00),v40,z0,tPen\WObj:=wPaper;
    MoveL Offs(pOrigin,202.19,197.10,0.00),v40,fine,tPen\WObj:=wPaper;
    MoveL Offs(pOrigin,202.19,197.10,6.00),v60,z5,tPen\WObj:=wPaper;
    MoveL Offs(pOrigin,210.48,204.32,6.00),vTravel,z5,tPen\WObj:=wPaper;
    MoveL Offs(pOrigin,210.48,204.32,0.00),v60,z0,tPen\WObj:=wPaper;
    MoveL Offs(pOrigin,211.32,205.18,0.00),v40,z0,tPen\WObj:=wPaper;
    MoveL Offs(pOrigin,210.48,204.32,0.00),v40,fine,tPen\WObj:=wPaper;
    MoveL Offs(pOrigin,210.48,204.32,6.00),v60,z5,tPen\WObj:=wPaper;
    MoveL Offs(pOrigin,209.62,206.02,6.00),vTravel,z5,tPen\WObj:=wPaper;
    MoveL Offs(pOrigin,209.62,206.02,0.00),v60,z0,tPen\WObj:=wPaper;
    MoveL Offs(pOrigin,209.20,204.96,0.00),v40,z0,tPen\WObj:=wPaper;
    MoveL Offs(pOrigin,196.24,189.66,0.00),v40,z0,tPen\WObj:=wPaper;
    MoveL Offs(pOrigin,197.09,188.74,0.00),v40,z0,tPen\WObj:=wPaper;
    MoveL Offs(pOrigin,206.44,185.41,0.00),v40,z0,tPen\WObj:=wPaper;
    MoveL Offs(pOrigin,206.58,184.77,0.00),v40,z0,tPen\WObj:=wPaper;
    MoveL Offs(pOrigin,194.11,177.98,0.00),v40,z0,tPen\WObj:=wPaper;
    MoveL Offs(pOrigin,193.69,177.34,0.00),v40,z0,tPen\WObj:=wPaper;
    MoveL Offs(pOrigin,200.27,151.62,0.00),v40,z0,tPen\WObj:=wPaper;
    MoveL Offs(pOrigin,205.59,132.50,0.00),v40,z0,tPen\WObj:=wPaper;
    MoveL Offs(pOrigin,206.86,125.28,0.00),v40,z0,tPen\WObj:=wPaper;
    MoveL Offs(pOrigin,207.71,123.36,0.00),v40,z0,tPen\WObj:=wPaper;
    MoveL Offs(pOrigin,208.14,120.60,0.00),v40,z0,tPen\WObj:=wPaper;
    MoveL Offs(pOrigin,208.14,120.60,0.00),v40,z0,tPen\WObj:=wPaper;
    MoveL Offs(pOrigin,209.13,119.96,0.00),v40,z0,tPen\WObj:=wPaper;
    MoveL Offs(pOrigin,211.75,110.61,0.00),v40,z0,tPen\WObj:=wPaper;
    MoveL Offs(pOrigin,213.88,101.69,0.00),v40,z0,tPen\WObj:=wPaper;
    MoveL Offs(pOrigin,215.36,93.40,0.00),v40,z0,tPen\WObj:=wPaper;
    MoveL Offs(pOrigin,216.64,80.01,0.00),v40,z0,tPen\WObj:=wPaper;
    MoveL Offs(pOrigin,216.64,68.96,0.00),v40,z0,tPen\WObj:=wPaper;
    MoveL Offs(pOrigin,216.21,68.54,0.00),v40,z0,tPen\WObj:=wPaper;
    MoveL Offs(pOrigin,216.21,68.54,0.00),v40,z0,tPen\WObj:=wPaper;
    MoveL Offs(pOrigin,216.00,64.93,0.00),v40,z0,tPen\WObj:=wPaper;
    MoveL Offs(pOrigin,216.21,63.86,0.00),v40,fine,tPen\WObj:=wPaper;
    MoveL Offs(pOrigin,216.21,63.86,6.00),v60,z5,tPen\WObj:=wPaper;
    MoveL Offs(pOrigin,213.66,62.80,6.00),vTravel,z5,tPen\WObj:=wPaper;
    MoveL Offs(pOrigin,213.66,62.80,0.00),v60,z0,tPen\WObj:=wPaper;
    MoveL Offs(pOrigin,213.24,63.22,0.00),v40,z0,tPen\WObj:=wPaper;
    MoveL Offs(pOrigin,213.66,62.80,0.00),v40,fine,tPen\WObj:=wPaper;
    MoveL Offs(pOrigin,213.66,62.80,6.00),v60,z5,tPen\WObj:=wPaper;
    MoveL Offs(pOrigin,217.49,58.76,6.00),vTravel,z5,tPen\WObj:=wPaper;
    MoveL Offs(pOrigin,217.49,58.76,0.00),v60,z0,tPen\WObj:=wPaper;
    MoveL Offs(pOrigin,217.27,59.19,0.00),v40,z0,tPen\WObj:=wPaper;
    MoveL Offs(pOrigin,217.49,58.76,0.00),v40,fine,tPen\WObj:=wPaper;
    MoveL Offs(pOrigin,217.49,58.76,6.00),v60,z5,tPen\WObj:=wPaper;
    MoveL Offs(pOrigin,216.43,57.70,6.00),vTravel,z5,tPen\WObj:=wPaper;
    MoveL Offs(pOrigin,216.43,57.70,0.00),v60,z0,tPen\WObj:=wPaper;
    MoveL Offs(pOrigin,216.21,58.12,0.00),v40,z0,tPen\WObj:=wPaper;
    MoveL Offs(pOrigin,216.43,57.70,0.00),v40,fine,tPen\WObj:=wPaper;
    MoveL Offs(pOrigin,216.43,57.70,6.00),v60,z5,tPen\WObj:=wPaper;
    MoveL Offs(pOrigin,215.79,53.88,6.00),vTravel,z5,tPen\WObj:=wPaper;
    MoveL Offs(pOrigin,215.79,53.88,0.00),v60,z0,tPen\WObj:=wPaper;
    MoveL Offs(pOrigin,216.21,54.30,0.00),v40,z0,tPen\WObj:=wPaper;
    MoveL Offs(pOrigin,215.79,53.88,0.00),v40,fine,tPen\WObj:=wPaper;
    MoveL Offs(pOrigin,215.79,53.88,6.00),v60,z5,tPen\WObj:=wPaper;
    MoveL Offs(pOrigin,218.98,52.81,6.00),vTravel,z5,tPen\WObj:=wPaper;
    MoveL Offs(pOrigin,218.98,52.81,0.00),v60,z0,tPen\WObj:=wPaper;
    MoveL Offs(pOrigin,217.91,53.88,0.00),v40,z0,tPen\WObj:=wPaper;
    MoveL Offs(pOrigin,218.98,52.81,0.00),v40,z0,tPen\WObj:=wPaper;
    MoveL Offs(pOrigin,219.61,52.17,0.00),v40,z0,tPen\WObj:=wPaper;
    MoveL Offs(pOrigin,219.19,52.60,0.00),v40,z0,tPen\WObj:=wPaper;
    MoveL Offs(pOrigin,219.61,52.17,0.00),v40,fine,tPen\WObj:=wPaper;
    MoveL Offs(pOrigin,219.61,52.17,6.00),v60,z5,tPen\WObj:=wPaper;
    MoveL Offs(pOrigin,227.26,65.14,6.00),vTravel,z5,tPen\WObj:=wPaper;
    MoveL Offs(pOrigin,227.26,65.14,0.00),v60,z0,tPen\WObj:=wPaper;
    MoveL Offs(pOrigin,227.83,64.93,0.00),v40,z0,tPen\WObj:=wPaper;
    MoveL Offs(pOrigin,230.45,61.31,0.00),v40,z0,tPen\WObj:=wPaper;
    MoveL Offs(pOrigin,236.61,51.54,0.00),v40,fine,tPen\WObj:=wPaper;
    MoveL Offs(pOrigin,236.61,51.54,6.00),v60,z5,tPen\WObj:=wPaper;
    MoveL Offs(pOrigin,237.25,61.10,6.00),vTravel,z5,tPen\WObj:=wPaper;
    MoveL Offs(pOrigin,237.25,61.10,0.00),v60,z0,tPen\WObj:=wPaper;
    MoveL Offs(pOrigin,235.76,62.80,0.00),v40,z0,tPen\WObj:=wPaper;
    MoveL Offs(pOrigin,233.00,64.78,0.00),v40,z0,tPen\WObj:=wPaper;
    MoveL Offs(pOrigin,228.75,66.91,0.00),v40,z0,tPen\WObj:=wPaper;
    MoveL Offs(pOrigin,227.69,67.05,0.00),v40,z0,tPen\WObj:=wPaper;
    MoveL Offs(pOrigin,227.69,67.05,0.00),v40,z0,tPen\WObj:=wPaper;
    MoveL Offs(pOrigin,230.24,81.29,0.00),v40,z0,tPen\WObj:=wPaper;
    MoveL Offs(pOrigin,230.88,82.14,0.00),v40,fine,tPen\WObj:=wPaper;
    MoveL Offs(pOrigin,230.88,82.14,6.00),v60,z5,tPen\WObj:=wPaper;
    MoveL Offs(pOrigin,232.57,78.95,6.00),vTravel,z5,tPen\WObj:=wPaper;
    MoveL Offs(pOrigin,232.57,78.95,0.00),v60,z0,tPen\WObj:=wPaper;
    MoveL Offs(pOrigin,232.36,79.38,0.00),v40,z0,tPen\WObj:=wPaper;
    MoveL Offs(pOrigin,232.57,78.95,0.00),v40,fine,tPen\WObj:=wPaper;
    MoveL Offs(pOrigin,232.57,78.95,6.00),v60,z5,tPen\WObj:=wPaper;
    MoveL Offs(pOrigin,233.21,77.89,6.00),vTravel,z5,tPen\WObj:=wPaper;
    MoveL Offs(pOrigin,233.21,77.89,0.00),v60,z0,tPen\WObj:=wPaper;
    MoveL Offs(pOrigin,233.00,78.31,0.00),v40,z0,tPen\WObj:=wPaper;
    MoveL Offs(pOrigin,233.21,77.89,0.00),v40,fine,tPen\WObj:=wPaper;
    MoveL Offs(pOrigin,233.21,77.89,6.00),v60,z5,tPen\WObj:=wPaper;
    MoveL Offs(pOrigin,227.69,67.05,6.00),vTravel,z5,tPen\WObj:=wPaper;
    MoveL Offs(pOrigin,227.69,67.05,0.00),v60,z0,tPen\WObj:=wPaper;
    MoveL Offs(pOrigin,227.26,66.62,0.00),v40,z0,tPen\WObj:=wPaper;
    MoveL Offs(pOrigin,227.26,65.14,0.00),v40,z0,tPen\WObj:=wPaper;
    MoveL Offs(pOrigin,227.26,65.14,0.00),v40,z0,tPen\WObj:=wPaper;
    MoveL Offs(pOrigin,226.84,64.50,0.00),v40,z0,tPen\WObj:=wPaper;
    MoveL Offs(pOrigin,222.45,49.41,0.00),v40,z0,tPen\WObj:=wPaper;
    MoveL Offs(pOrigin,227.69,41.41,0.00),v40,z0,tPen\WObj:=wPaper;
    MoveL Offs(pOrigin,237.68,40.49,0.00),v40,z0,tPen\WObj:=wPaper;
    MoveL Offs(pOrigin,238.74,40.91,0.00),v40,fine,tPen\WObj:=wPaper;
  ENDPROC

  PROC DrawPart77()
    MoveL Offs(pOrigin,238.74,40.91,6.00),v60,z5,tPen\WObj:=wPaper;
    MoveL Offs(pOrigin,245.96,31.99,6.00),vTravel,z5,tPen\WObj:=wPaper;
    MoveL Offs(pOrigin,245.96,31.99,0.00),v60,z0,tPen\WObj:=wPaper;
    MoveL Offs(pOrigin,245.75,32.41,0.00),v40,z0,tPen\WObj:=wPaper;
    MoveL Offs(pOrigin,245.96,31.99,0.00),v40,z0,tPen\WObj:=wPaper;
    MoveL Offs(pOrigin,245.11,31.35,0.00),v40,z0,tPen\WObj:=wPaper;
    MoveL Offs(pOrigin,245.32,30.92,0.00),v40,z0,tPen\WObj:=wPaper;
    MoveL Offs(pOrigin,245.11,31.35,0.00),v40,fine,tPen\WObj:=wPaper;
    MoveL Offs(pOrigin,245.11,31.35,6.00),v60,z5,tPen\WObj:=wPaper;
    MoveL Offs(pOrigin,245.75,27.95,6.00),vTravel,z5,tPen\WObj:=wPaper;
    MoveL Offs(pOrigin,245.75,27.95,0.00),v60,z0,tPen\WObj:=wPaper;
    MoveL Offs(pOrigin,214.51,21.08,0.00),v40,z0,tPen\WObj:=wPaper;
    MoveL Offs(pOrigin,214.09,20.51,0.00),v40,z0,tPen\WObj:=wPaper;
    MoveL Offs(pOrigin,214.09,20.51,0.00),v40,z0,tPen\WObj:=wPaper;
    MoveL Offs(pOrigin,214.94,20.09,0.00),v40,z0,tPen\WObj:=wPaper;
    MoveL Offs(pOrigin,233.64,18.39,0.00),v40,z0,tPen\WObj:=wPaper;
    MoveL Offs(pOrigin,271.67,27.81,0.00),v40,z0,tPen\WObj:=wPaper;
    MoveL Offs(pOrigin,272.10,28.59,0.00),v40,z0,tPen\WObj:=wPaper;
    MoveL Offs(pOrigin,272.10,28.59,0.00),v40,z0,tPen\WObj:=wPaper;
    MoveL Offs(pOrigin,269.12,28.59,0.00),v40,z0,tPen\WObj:=wPaper;
    MoveL Offs(pOrigin,264.88,27.74,0.00),v40,z0,tPen\WObj:=wPaper;
    MoveL Offs(pOrigin,258.08,27.74,0.00),v40,z0,tPen\WObj:=wPaper;
    MoveL Offs(pOrigin,256.16,28.30,0.00),v40,z0,tPen\WObj:=wPaper;
    MoveL Offs(pOrigin,254.46,29.51,0.00),v40,z0,tPen\WObj:=wPaper;
    MoveL Offs(pOrigin,252.12,29.30,0.00),v40,z0,tPen\WObj:=wPaper;
    MoveL Offs(pOrigin,251.91,30.08,0.00),v40,z0,tPen\WObj:=wPaper;
    MoveL Offs(pOrigin,251.91,30.08,0.00),v40,z0,tPen\WObj:=wPaper;
    MoveL Offs(pOrigin,251.06,30.08,0.00),v40,z0,tPen\WObj:=wPaper;
    MoveL Offs(pOrigin,250.64,29.44,0.00),v40,z0,tPen\WObj:=wPaper;
    MoveL Offs(pOrigin,250.64,29.44,0.00),v40,z0,tPen\WObj:=wPaper;
    MoveL Offs(pOrigin,251.06,29.01,0.00),v40,z0,tPen\WObj:=wPaper;
    MoveL Offs(pOrigin,251.91,29.23,0.00),v40,fine,tPen\WObj:=wPaper;
    MoveL Offs(pOrigin,251.91,29.23,6.00),v60,z5,tPen\WObj:=wPaper;
    MoveL Offs(pOrigin,250.00,31.56,6.00),vTravel,z5,tPen\WObj:=wPaper;
    MoveL Offs(pOrigin,250.00,31.56,0.00),v60,z0,tPen\WObj:=wPaper;
    MoveL Offs(pOrigin,247.66,31.14,0.00),v40,z0,tPen\WObj:=wPaper;
    MoveL Offs(pOrigin,246.39,31.63,0.00),v40,z0,tPen\WObj:=wPaper;
    MoveL Offs(pOrigin,245.54,32.84,0.00),v40,z0,tPen\WObj:=wPaper;
    MoveL Offs(pOrigin,245.32,34.75,0.00),v40,z0,tPen\WObj:=wPaper;
    MoveL Offs(pOrigin,245.82,35.95,0.00),v40,z0,tPen\WObj:=wPaper;
    MoveL Offs(pOrigin,248.30,37.94,0.00),v40,z0,tPen\WObj:=wPaper;
    MoveL Offs(pOrigin,248.80,39.00,0.00),v40,z0,tPen\WObj:=wPaper;
    MoveL Offs(pOrigin,250.21,40.28,0.00),v40,z0,tPen\WObj:=wPaper;
    MoveL Offs(pOrigin,259.35,47.08,0.00),v40,z0,tPen\WObj:=wPaper;
    MoveL Offs(pOrigin,265.30,50.97,0.00),v40,z0,tPen\WObj:=wPaper;
    MoveL Offs(pOrigin,269.34,52.88,0.00),v40,z0,tPen\WObj:=wPaper;
    MoveL Offs(pOrigin,278.48,56.28,0.00),v40,z0,tPen\WObj:=wPaper;
    MoveL Offs(pOrigin,279.54,56.92,0.00),v40,z0,tPen\WObj:=wPaper;
    MoveL Offs(pOrigin,279.96,57.70,0.00),v40,z0,tPen\WObj:=wPaper;
    MoveL Offs(pOrigin,279.96,57.70,0.00),v40,z0,tPen\WObj:=wPaper;
    MoveL Offs(pOrigin,281.66,58.83,0.00),v40,z0,tPen\WObj:=wPaper;
    MoveL Offs(pOrigin,283.15,60.46,0.00),v40,fine,tPen\WObj:=wPaper;
    MoveL Offs(pOrigin,283.15,60.46,6.00),v60,z5,tPen\WObj:=wPaper;
    MoveL Offs(pOrigin,279.96,57.70,6.00),vTravel,z5,tPen\WObj:=wPaper;
    MoveL Offs(pOrigin,279.96,57.70,0.00),v60,z0,tPen\WObj:=wPaper;
    MoveL Offs(pOrigin,274.86,56.00,0.00),v40,z0,tPen\WObj:=wPaper;
    MoveL Offs(pOrigin,274.37,56.21,0.00),v40,z0,tPen\WObj:=wPaper;
    MoveL Offs(pOrigin,274.01,57.06,0.00),v40,z0,tPen\WObj:=wPaper;
    MoveL Offs(pOrigin,272.95,57.49,0.00),v40,z0,tPen\WObj:=wPaper;
    MoveL Offs(pOrigin,272.95,57.49,0.00),v40,z0,tPen\WObj:=wPaper;
    MoveL Offs(pOrigin,272.67,55.58,0.00),v40,z0,tPen\WObj:=wPaper;
    MoveL Offs(pOrigin,271.04,55.43,0.00),v40,z0,tPen\WObj:=wPaper;
    MoveL Offs(pOrigin,268.06,60.46,0.00),v40,z0,tPen\WObj:=wPaper;
    MoveL Offs(pOrigin,268.06,60.46,0.00),v40,z0,tPen\WObj:=wPaper;
    MoveL Offs(pOrigin,265.09,60.11,0.00),v40,z0,tPen\WObj:=wPaper;
    MoveL Offs(pOrigin,259.35,56.85,0.00),v40,z0,tPen\WObj:=wPaper;
    MoveL Offs(pOrigin,250.85,48.78,0.00),v40,z0,tPen\WObj:=wPaper;
    MoveL Offs(pOrigin,246.18,43.46,0.00),v40,z0,tPen\WObj:=wPaper;
    MoveL Offs(pOrigin,245.61,42.19,0.00),v40,z0,tPen\WObj:=wPaper;
    MoveL Offs(pOrigin,247.24,41.34,0.00),v40,z0,tPen\WObj:=wPaper;
    MoveL Offs(pOrigin,248.09,40.35,0.00),v40,z0,tPen\WObj:=wPaper;
    MoveL Offs(pOrigin,248.51,40.42,0.00),v40,z0,tPen\WObj:=wPaper;
    MoveL Offs(pOrigin,260.20,49.20,0.00),v40,z0,tPen\WObj:=wPaper;
    MoveL Offs(pOrigin,264.66,52.03,0.00),v40,z0,tPen\WObj:=wPaper;
    MoveL Offs(pOrigin,269.55,54.16,0.00),v40,z0,tPen\WObj:=wPaper;
    MoveL Offs(pOrigin,270.61,55.58,0.00),v40,fine,tPen\WObj:=wPaper;
    MoveL Offs(pOrigin,270.61,55.58,6.00),v60,z5,tPen\WObj:=wPaper;
    MoveL Offs(pOrigin,269.76,57.49,6.00),vTravel,z5,tPen\WObj:=wPaper;
    MoveL Offs(pOrigin,269.76,57.49,0.00),v60,z0,tPen\WObj:=wPaper;
    MoveL Offs(pOrigin,269.55,57.91,0.00),v40,z0,tPen\WObj:=wPaper;
    MoveL Offs(pOrigin,269.76,57.49,0.00),v40,fine,tPen\WObj:=wPaper;
    MoveL Offs(pOrigin,269.76,57.49,6.00),v60,z5,tPen\WObj:=wPaper;
    MoveL Offs(pOrigin,272.31,58.76,6.00),vTravel,z5,tPen\WObj:=wPaper;
    MoveL Offs(pOrigin,272.31,58.76,0.00),v60,z0,tPen\WObj:=wPaper;
    MoveL Offs(pOrigin,272.10,59.19,0.00),v40,z0,tPen\WObj:=wPaper;
    MoveL Offs(pOrigin,272.31,58.76,0.00),v40,fine,tPen\WObj:=wPaper;
    MoveL Offs(pOrigin,272.31,58.76,6.00),v60,z5,tPen\WObj:=wPaper;
    MoveL Offs(pOrigin,272.95,57.49,6.00),vTravel,z5,tPen\WObj:=wPaper;
    MoveL Offs(pOrigin,272.95,57.49,0.00),v60,z0,tPen\WObj:=wPaper;
    MoveL Offs(pOrigin,271.04,61.10,0.00),v40,fine,tPen\WObj:=wPaper;
    MoveL Offs(pOrigin,271.04,61.10,6.00),v60,z5,tPen\WObj:=wPaper;
    MoveL Offs(pOrigin,272.74,55.36,6.00),vTravel,z5,tPen\WObj:=wPaper;
    MoveL Offs(pOrigin,272.74,55.36,0.00),v60,z0,tPen\WObj:=wPaper;
    MoveL Offs(pOrigin,272.95,55.79,0.00),v40,z0,tPen\WObj:=wPaper;
    MoveL Offs(pOrigin,272.74,55.36,0.00),v40,fine,tPen\WObj:=wPaper;
    MoveL Offs(pOrigin,272.74,55.36,6.00),v60,z5,tPen\WObj:=wPaper;
    MoveL Offs(pOrigin,268.06,49.20,6.00),vTravel,z5,tPen\WObj:=wPaper;
    MoveL Offs(pOrigin,268.06,49.20,0.00),v60,z0,tPen\WObj:=wPaper;
    MoveL Offs(pOrigin,269.62,47.08,0.00),v40,z0,tPen\WObj:=wPaper;
    MoveL Offs(pOrigin,269.76,45.80,0.00),v40,fine,tPen\WObj:=wPaper;
    MoveL Offs(pOrigin,269.76,45.80,6.00),v60,z5,tPen\WObj:=wPaper;
    MoveL Offs(pOrigin,267.00,44.10,6.00),vTravel,z5,tPen\WObj:=wPaper;
    MoveL Offs(pOrigin,267.00,44.10,0.00),v60,z0,tPen\WObj:=wPaper;
    MoveL Offs(pOrigin,266.15,44.95,0.00),v40,z0,tPen\WObj:=wPaper;
    MoveL Offs(pOrigin,265.30,46.65,0.00),v40,fine,tPen\WObj:=wPaper;
    MoveL Offs(pOrigin,265.30,46.65,6.00),v60,z5,tPen\WObj:=wPaper;
    MoveL Offs(pOrigin,276.35,38.36,6.00),vTravel,z5,tPen\WObj:=wPaper;
    MoveL Offs(pOrigin,276.35,38.36,0.00),v60,z0,tPen\WObj:=wPaper;
    MoveL Offs(pOrigin,276.35,37.72,0.00),v40,z0,tPen\WObj:=wPaper;
    MoveL Offs(pOrigin,277.20,36.24,0.00),v40,fine,tPen\WObj:=wPaper;
    MoveL Offs(pOrigin,277.20,36.24,6.00),v60,z5,tPen\WObj:=wPaper;
    MoveL Offs(pOrigin,284.42,33.69,6.00),vTravel,z5,tPen\WObj:=wPaper;
    MoveL Offs(pOrigin,284.42,33.69,0.00),v60,z0,tPen\WObj:=wPaper;
    MoveL Offs(pOrigin,284.85,33.90,0.00),v40,z0,tPen\WObj:=wPaper;
    MoveL Offs(pOrigin,284.42,33.69,0.00),v40,fine,tPen\WObj:=wPaper;
    MoveL Offs(pOrigin,284.42,33.69,6.00),v60,z5,tPen\WObj:=wPaper;
    MoveL Offs(pOrigin,286.98,41.34,6.00),vTravel,z5,tPen\WObj:=wPaper;
    MoveL Offs(pOrigin,286.98,41.34,0.00),v60,z0,tPen\WObj:=wPaper;
    MoveL Offs(pOrigin,287.61,41.97,0.00),v40,fine,tPen\WObj:=wPaper;
    MoveL Offs(pOrigin,287.61,41.97,6.00),v60,z5,tPen\WObj:=wPaper;
  ENDPROC

  PROC DrawPart78()
    MoveL Offs(pOrigin,301.42,49.41,6.00),vTravel,z5,tPen\WObj:=wPaper;
    MoveL Offs(pOrigin,301.42,49.41,0.00),v60,z0,tPen\WObj:=wPaper;
    MoveL Offs(pOrigin,303.12,43.89,0.00),v40,z0,tPen\WObj:=wPaper;
    MoveL Offs(pOrigin,303.76,39.85,0.00),v40,fine,tPen\WObj:=wPaper;
    MoveL Offs(pOrigin,303.76,39.85,6.00),v60,z5,tPen\WObj:=wPaper;
    MoveL Offs(pOrigin,305.89,45.16,6.00),vTravel,z5,tPen\WObj:=wPaper;
    MoveL Offs(pOrigin,305.89,45.16,0.00),v60,z0,tPen\WObj:=wPaper;
    MoveL Offs(pOrigin,305.89,46.44,0.00),v40,z0,tPen\WObj:=wPaper;
    MoveL Offs(pOrigin,304.26,50.90,0.00),v40,z0,tPen\WObj:=wPaper;
    MoveL Offs(pOrigin,302.63,53.88,0.00),v40,z0,tPen\WObj:=wPaper;
    MoveL Offs(pOrigin,300.15,57.06,0.00),v40,fine,tPen\WObj:=wPaper;
    MoveL Offs(pOrigin,300.15,57.06,6.00),v60,z5,tPen\WObj:=wPaper;
    MoveL Offs(pOrigin,296.96,56.85,6.00),vTravel,z5,tPen\WObj:=wPaper;
    MoveL Offs(pOrigin,296.96,56.85,0.00),v60,z0,tPen\WObj:=wPaper;
    MoveL Offs(pOrigin,296.33,57.91,0.00),v40,z0,tPen\WObj:=wPaper;
    MoveL Offs(pOrigin,292.29,61.74,0.00),v40,fine,tPen\WObj:=wPaper;
    MoveL Offs(pOrigin,292.29,61.74,6.00),v60,z5,tPen\WObj:=wPaper;
    MoveL Offs(pOrigin,294.62,64.07,6.00),vTravel,z5,tPen\WObj:=wPaper;
    MoveL Offs(pOrigin,294.62,64.07,0.00),v60,z0,tPen\WObj:=wPaper;
    MoveL Offs(pOrigin,292.92,64.36,0.00),v40,z0,tPen\WObj:=wPaper;
    MoveL Offs(pOrigin,290.59,65.56,0.00),v40,z0,tPen\WObj:=wPaper;
    MoveL Offs(pOrigin,289.95,65.78,0.00),v40,z0,tPen\WObj:=wPaper;
    MoveL Offs(pOrigin,286.76,67.69,0.00),v40,z0,tPen\WObj:=wPaper;
    MoveL Offs(pOrigin,286.55,69.81,0.00),v40,z0,tPen\WObj:=wPaper;
    MoveL Offs(pOrigin,288.25,80.44,0.00),v40,z0,tPen\WObj:=wPaper;
    MoveL Offs(pOrigin,291.30,93.82,0.00),v40,z0,tPen\WObj:=wPaper;
    MoveL Offs(pOrigin,292.08,94.46,0.00),v40,fine,tPen\WObj:=wPaper;
    MoveL Offs(pOrigin,292.08,94.46,6.00),v60,z5,tPen\WObj:=wPaper;
    MoveL Offs(pOrigin,296.11,105.30,6.00),vTravel,z5,tPen\WObj:=wPaper;
    MoveL Offs(pOrigin,296.11,105.30,0.00),v60,z0,tPen\WObj:=wPaper;
    MoveL Offs(pOrigin,294.27,104.88,0.00),v40,z0,tPen\WObj:=wPaper;
    MoveL Offs(pOrigin,293.14,100.84,0.00),v40,z0,tPen\WObj:=wPaper;
    MoveL Offs(pOrigin,292.29,96.59,0.00),v40,z0,tPen\WObj:=wPaper;
    MoveL Offs(pOrigin,291.86,82.78,0.00),v40,z0,tPen\WObj:=wPaper;
    MoveL Offs(pOrigin,292.50,75.34,0.00),v40,z0,tPen\WObj:=wPaper;
    MoveL Offs(pOrigin,293.77,67.90,0.00),v40,z0,tPen\WObj:=wPaper;
    MoveL Offs(pOrigin,295.05,63.65,0.00),v40,z0,tPen\WObj:=wPaper;
    MoveL Offs(pOrigin,298.24,62.80,0.00),v40,z0,tPen\WObj:=wPaper;
    MoveL Offs(pOrigin,301.21,64.85,0.00),v40,z0,tPen\WObj:=wPaper;
    MoveL Offs(pOrigin,304.83,66.20,0.00),v40,z0,tPen\WObj:=wPaper;
    MoveL Offs(pOrigin,310.14,67.40,0.00),v40,z0,tPen\WObj:=wPaper;
    MoveL Offs(pOrigin,314.17,69.95,0.00),v40,z0,tPen\WObj:=wPaper;
    MoveL Offs(pOrigin,316.73,70.95,0.00),v40,z0,tPen\WObj:=wPaper;
    MoveL Offs(pOrigin,322.46,72.57,0.00),v40,z0,tPen\WObj:=wPaper;
    MoveL Offs(pOrigin,333.30,74.49,0.00),v40,z0,tPen\WObj:=wPaper;
    MoveL Offs(pOrigin,334.15,74.91,0.00),v40,z0,tPen\WObj:=wPaper;
    MoveL Offs(pOrigin,334.15,74.91,0.00),v40,z0,tPen\WObj:=wPaper;
    MoveL Offs(pOrigin,340.17,88.09,0.00),v40,z0,tPen\WObj:=wPaper;
    MoveL Offs(pOrigin,342.01,92.97,0.00),v40,fine,tPen\WObj:=wPaper;
    MoveL Offs(pOrigin,342.01,92.97,6.00),v60,z5,tPen\WObj:=wPaper;
    MoveL Offs(pOrigin,347.11,97.01,6.00),vTravel,z5,tPen\WObj:=wPaper;
    MoveL Offs(pOrigin,347.11,97.01,0.00),v60,z0,tPen\WObj:=wPaper;
    MoveL Offs(pOrigin,347.33,99.56,0.00),v40,fine,tPen\WObj:=wPaper;
    MoveL Offs(pOrigin,347.33,99.56,6.00),v60,z5,tPen\WObj:=wPaper;
    MoveL Offs(pOrigin,346.26,101.05,6.00),vTravel,z5,tPen\WObj:=wPaper;
    MoveL Offs(pOrigin,346.26,101.05,0.00),v60,z0,tPen\WObj:=wPaper;
    MoveL Offs(pOrigin,346.48,100.41,0.00),v40,z0,tPen\WObj:=wPaper;
    MoveL Offs(pOrigin,344.14,91.91,0.00),v40,z0,tPen\WObj:=wPaper;
    MoveL Offs(pOrigin,339.82,80.65,0.00),v40,z0,tPen\WObj:=wPaper;
    MoveL Offs(pOrigin,339.67,79.38,0.00),v40,fine,tPen\WObj:=wPaper;
    MoveL Offs(pOrigin,339.67,79.38,6.00),v60,z5,tPen\WObj:=wPaper;
    MoveL Offs(pOrigin,337.98,75.76,6.00),vTravel,z5,tPen\WObj:=wPaper;
    MoveL Offs(pOrigin,337.98,75.76,0.00),v60,z0,tPen\WObj:=wPaper;
    MoveL Offs(pOrigin,339.04,75.34,0.00),v40,z0,tPen\WObj:=wPaper;
    MoveL Offs(pOrigin,346.26,76.40,0.00),v40,z0,tPen\WObj:=wPaper;
    MoveL Offs(pOrigin,346.90,76.82,0.00),v40,z0,tPen\WObj:=wPaper;
    MoveL Offs(pOrigin,348.17,84.26,0.00),v40,z0,tPen\WObj:=wPaper;
    MoveL Offs(pOrigin,348.81,92.76,0.00),v40,z0,tPen\WObj:=wPaper;
    MoveL Offs(pOrigin,348.46,94.68,0.00),v40,z0,tPen\WObj:=wPaper;
    MoveL Offs(pOrigin,347.11,97.01,0.00),v40,z0,tPen\WObj:=wPaper;
    MoveL Offs(pOrigin,347.11,97.01,0.00),v40,z0,tPen\WObj:=wPaper;
    MoveL Offs(pOrigin,342.30,83.84,0.00),v40,z0,tPen\WObj:=wPaper;
    MoveL Offs(pOrigin,340.45,79.80,0.00),v40,z0,tPen\WObj:=wPaper;
    MoveL Offs(pOrigin,339.39,78.74,0.00),v40,z0,tPen\WObj:=wPaper;
    MoveL Offs(pOrigin,337.98,75.76,0.00),v40,z0,tPen\WObj:=wPaper;
    MoveL Offs(pOrigin,337.98,75.76,0.00),v40,z0,tPen\WObj:=wPaper;
    MoveL Offs(pOrigin,336.06,74.91,0.00),v40,z0,tPen\WObj:=wPaper;
    MoveL Offs(pOrigin,334.58,74.70,0.00),v40,z0,tPen\WObj:=wPaper;
    MoveL Offs(pOrigin,334.15,74.91,0.00),v40,fine,tPen\WObj:=wPaper;
    MoveL Offs(pOrigin,334.15,74.91,6.00),v60,z5,tPen\WObj:=wPaper;
    MoveL Offs(pOrigin,339.46,72.79,6.00),vTravel,z5,tPen\WObj:=wPaper;
    MoveL Offs(pOrigin,339.46,72.79,0.00),v60,z0,tPen\WObj:=wPaper;
    MoveL Offs(pOrigin,342.44,72.79,0.00),v40,z0,tPen\WObj:=wPaper;
    MoveL Offs(pOrigin,347.33,72.15,0.00),v40,z0,tPen\WObj:=wPaper;
    MoveL Offs(pOrigin,353.06,70.88,0.00),v40,z0,tPen\WObj:=wPaper;
    MoveL Offs(pOrigin,358.80,69.03,0.00),v40,z0,tPen\WObj:=wPaper;
    MoveL Offs(pOrigin,363.05,67.33,0.00),v40,z0,tPen\WObj:=wPaper;
    MoveL Offs(pOrigin,368.79,64.36,0.00),v40,z0,tPen\WObj:=wPaper;
    MoveL Offs(pOrigin,373.25,61.53,0.00),v40,z0,tPen\WObj:=wPaper;
    MoveL Offs(pOrigin,376.65,58.76,0.00),v40,z0,tPen\WObj:=wPaper;
    MoveL Offs(pOrigin,377.08,58.55,0.00),v40,z0,tPen\WObj:=wPaper;
    MoveL Offs(pOrigin,384.73,50.90,0.00),v40,fine,tPen\WObj:=wPaper;
    MoveL Offs(pOrigin,384.73,50.90,6.00),v60,z5,tPen\WObj:=wPaper;
    MoveL Offs(pOrigin,382.39,48.14,6.00),vTravel,z5,tPen\WObj:=wPaper;
    MoveL Offs(pOrigin,382.39,48.14,0.00),v60,z0,tPen\WObj:=wPaper;
    MoveL Offs(pOrigin,381.75,48.78,0.00),v40,z0,tPen\WObj:=wPaper;
    MoveL Offs(pOrigin,382.39,48.14,0.00),v40,fine,tPen\WObj:=wPaper;
    MoveL Offs(pOrigin,382.39,48.14,6.00),v60,z5,tPen\WObj:=wPaper;
    MoveL Offs(pOrigin,384.09,46.44,6.00),vTravel,z5,tPen\WObj:=wPaper;
    MoveL Offs(pOrigin,384.09,46.44,0.00),v60,z0,tPen\WObj:=wPaper;
    MoveL Offs(pOrigin,382.60,47.92,0.00),v40,z0,tPen\WObj:=wPaper;
    MoveL Offs(pOrigin,384.09,46.44,0.00),v40,fine,tPen\WObj:=wPaper;
    MoveL Offs(pOrigin,384.09,46.44,6.00),v60,z5,tPen\WObj:=wPaper;
    MoveL Offs(pOrigin,387.91,42.61,6.00),vTravel,z5,tPen\WObj:=wPaper;
    MoveL Offs(pOrigin,387.91,42.61,0.00),v60,z0,tPen\WObj:=wPaper;
    MoveL Offs(pOrigin,377.92,52.60,0.00),v40,z0,tPen\WObj:=wPaper;
    MoveL Offs(pOrigin,369.42,59.61,0.00),v40,fine,tPen\WObj:=wPaper;
    MoveL Offs(pOrigin,369.42,59.61,6.00),v60,z5,tPen\WObj:=wPaper;
    MoveL Offs(pOrigin,379.20,51.11,6.00),vTravel,z5,tPen\WObj:=wPaper;
    MoveL Offs(pOrigin,379.20,51.11,0.00),v60,z0,tPen\WObj:=wPaper;
    MoveL Offs(pOrigin,377.71,52.60,0.00),v40,z0,tPen\WObj:=wPaper;
    MoveL Offs(pOrigin,379.20,51.11,0.00),v40,fine,tPen\WObj:=wPaper;
    MoveL Offs(pOrigin,379.20,51.11,6.00),v60,z5,tPen\WObj:=wPaper;
    MoveL Offs(pOrigin,386.00,39.00,6.00),vTravel,z5,tPen\WObj:=wPaper;
    MoveL Offs(pOrigin,386.00,39.00,0.00),v60,z0,tPen\WObj:=wPaper;
    MoveL Offs(pOrigin,377.08,37.02,0.00),v40,z0,tPen\WObj:=wPaper;
    MoveL Offs(pOrigin,376.23,36.31,0.00),v40,z0,tPen\WObj:=wPaper;
    MoveL Offs(pOrigin,368.15,33.40,0.00),v40,z0,tPen\WObj:=wPaper;
    MoveL Offs(pOrigin,367.73,32.84,0.00),v40,z0,tPen\WObj:=wPaper;
    MoveL Offs(pOrigin,367.73,32.84,0.00),v40,z0,tPen\WObj:=wPaper;
  ENDPROC

  PROC DrawPart79()
    MoveL Offs(pOrigin,368.58,32.62,0.00),v40,z0,tPen\WObj:=wPaper;
    MoveL Offs(pOrigin,382.60,34.54,0.00),v40,z0,tPen\WObj:=wPaper;
    MoveL Offs(pOrigin,394.29,36.66,0.00),v40,z0,tPen\WObj:=wPaper;
    MoveL Offs(pOrigin,400.02,38.15,0.00),v40,z0,tPen\WObj:=wPaper;
    MoveL Offs(pOrigin,406.40,40.70,0.00),v40,z0,tPen\WObj:=wPaper;
    MoveL Offs(pOrigin,407.67,42.33,0.00),v40,z0,tPen\WObj:=wPaper;
    MoveL Offs(pOrigin,408.31,42.61,0.00),v40,z0,tPen\WObj:=wPaper;
    MoveL Offs(pOrigin,408.31,42.61,0.00),v40,z0,tPen\WObj:=wPaper;
    MoveL Offs(pOrigin,409.80,43.04,0.00),v40,z0,tPen\WObj:=wPaper;
    MoveL Offs(pOrigin,412.00,45.80,0.00),v40,z0,tPen\WObj:=wPaper;
    MoveL Offs(pOrigin,413.48,48.99,0.00),v40,z0,tPen\WObj:=wPaper;
    MoveL Offs(pOrigin,414.48,52.39,0.00),v40,z0,tPen\WObj:=wPaper;
    MoveL Offs(pOrigin,414.90,55.15,0.00),v40,z0,tPen\WObj:=wPaper;
    MoveL Offs(pOrigin,414.90,58.76,0.00),v40,z0,tPen\WObj:=wPaper;
    MoveL Offs(pOrigin,414.26,62.80,0.00),v40,z0,tPen\WObj:=wPaper;
    MoveL Offs(pOrigin,413.55,65.14,0.00),v40,z0,tPen\WObj:=wPaper;
    MoveL Offs(pOrigin,411.08,68.75,0.00),v40,z0,tPen\WObj:=wPaper;
    MoveL Offs(pOrigin,408.10,71.72,0.00),v40,z0,tPen\WObj:=wPaper;
    MoveL Offs(pOrigin,404.91,74.28,0.00),v40,z0,tPen\WObj:=wPaper;
    MoveL Offs(pOrigin,400.24,77.32,0.00),v40,z0,tPen\WObj:=wPaper;
    MoveL Offs(pOrigin,394.50,80.30,0.00),v40,z0,tPen\WObj:=wPaper;
    MoveL Offs(pOrigin,387.70,82.78,0.00),v40,z0,tPen\WObj:=wPaper;
    MoveL Offs(pOrigin,381.33,84.05,0.00),v40,z0,tPen\WObj:=wPaper;
    MoveL Offs(pOrigin,376.01,83.84,0.00),v40,z0,tPen\WObj:=wPaper;
    MoveL Offs(pOrigin,368.36,81.15,0.00),v40,z0,tPen\WObj:=wPaper;
    MoveL Offs(pOrigin,367.30,79.94,0.00),v40,z0,tPen\WObj:=wPaper;
    MoveL Offs(pOrigin,365.17,79.30,0.00),v40,z0,tPen\WObj:=wPaper;
    MoveL Offs(pOrigin,362.91,77.68,0.00),v40,z0,tPen\WObj:=wPaper;
    MoveL Offs(pOrigin,363.26,77.25,0.00),v40,z0,tPen\WObj:=wPaper;
    MoveL Offs(pOrigin,368.15,77.04,0.00),v40,z0,tPen\WObj:=wPaper;
    MoveL Offs(pOrigin,368.65,76.61,0.00),v40,z0,tPen\WObj:=wPaper;
    MoveL Offs(pOrigin,368.15,76.19,0.00),v40,z0,tPen\WObj:=wPaper;
    MoveL Offs(pOrigin,360.29,76.40,0.00),v40,z0,tPen\WObj:=wPaper;
    MoveL Offs(pOrigin,356.67,76.19,0.00),v40,z0,tPen\WObj:=wPaper;
    MoveL Offs(pOrigin,337.76,73.85,0.00),v40,z0,tPen\WObj:=wPaper;
    MoveL Offs(pOrigin,327.56,72.15,0.00),v40,z0,tPen\WObj:=wPaper;
    MoveL Offs(pOrigin,319.91,70.45,0.00),v40,z0,tPen\WObj:=wPaper;
    MoveL Offs(pOrigin,316.51,69.32,0.00),v40,z0,tPen\WObj:=wPaper;
    MoveL Offs(pOrigin,316.30,68.75,0.00),v40,z0,tPen\WObj:=wPaper;
    MoveL Offs(pOrigin,316.30,68.75,0.00),v40,z0,tPen\WObj:=wPaper;
    MoveL Offs(pOrigin,322.25,68.54,0.00),v40,z0,tPen\WObj:=wPaper;
    MoveL Offs(pOrigin,326.71,67.19,0.00),v40,z0,tPen\WObj:=wPaper;
    MoveL Offs(pOrigin,330.75,65.21,0.00),v40,z0,tPen\WObj:=wPaper;
    MoveL Offs(pOrigin,335.00,62.38,0.00),v40,z0,tPen\WObj:=wPaper;
    MoveL Offs(pOrigin,337.98,59.83,0.00),v40,z0,tPen\WObj:=wPaper;
    MoveL Offs(pOrigin,343.08,54.09,0.00),v40,z0,tPen\WObj:=wPaper;
    MoveL Offs(pOrigin,347.82,46.65,0.00),v40,z0,tPen\WObj:=wPaper;
    MoveL Offs(pOrigin,349.95,42.19,0.00),v40,z0,tPen\WObj:=wPaper;
    MoveL Offs(pOrigin,350.94,39.00,0.00),v40,z0,tPen\WObj:=wPaper;
    MoveL Offs(pOrigin,350.94,34.54,0.00),v40,z0,tPen\WObj:=wPaper;
    MoveL Offs(pOrigin,350.02,31.56,0.00),v40,z0,tPen\WObj:=wPaper;
    MoveL Offs(pOrigin,347.96,28.16,0.00),v40,z0,tPen\WObj:=wPaper;
    MoveL Offs(pOrigin,346.05,26.46,0.00),v40,z0,tPen\WObj:=wPaper;
    MoveL Offs(pOrigin,346.05,25.90,0.00),v40,z0,tPen\WObj:=wPaper;
    MoveL Offs(pOrigin,347.11,25.83,0.00),v40,z0,tPen\WObj:=wPaper;
    MoveL Offs(pOrigin,350.73,27.03,0.00),v40,z0,tPen\WObj:=wPaper;
    MoveL Offs(pOrigin,360.71,31.70,0.00),v40,z0,tPen\WObj:=wPaper;
    MoveL Offs(pOrigin,367.94,34.61,0.00),v40,z0,tPen\WObj:=wPaper;
    MoveL Offs(pOrigin,376.01,37.09,0.00),v40,z0,tPen\WObj:=wPaper;
    MoveL Offs(pOrigin,376.65,36.88,0.00),v40,fine,tPen\WObj:=wPaper;
    MoveL Offs(pOrigin,376.65,36.88,6.00),v60,z5,tPen\WObj:=wPaper;
    MoveL Offs(pOrigin,354.34,43.25,6.00),vTravel,z5,tPen\WObj:=wPaper;
    MoveL Offs(pOrigin,354.34,43.25,0.00),v60,z0,tPen\WObj:=wPaper;
    MoveL Offs(pOrigin,354.55,38.79,0.00),v40,z0,tPen\WObj:=wPaper;
    MoveL Offs(pOrigin,354.12,36.88,0.00),v40,z0,tPen\WObj:=wPaper;
    MoveL Offs(pOrigin,352.92,33.69,0.00),v40,z0,tPen\WObj:=wPaper;
    MoveL Offs(pOrigin,350.94,30.29,0.00),v40,fine,tPen\WObj:=wPaper;
    MoveL Offs(pOrigin,350.94,30.29,6.00),v60,z5,tPen\WObj:=wPaper;
    MoveL Offs(pOrigin,349.24,30.29,6.00),vTravel,z5,tPen\WObj:=wPaper;
    MoveL Offs(pOrigin,349.24,30.29,0.00),v60,z0,tPen\WObj:=wPaper;
    MoveL Offs(pOrigin,349.45,30.71,0.00),v40,z0,tPen\WObj:=wPaper;
    MoveL Offs(pOrigin,349.24,30.29,0.00),v40,fine,tPen\WObj:=wPaper;
    MoveL Offs(pOrigin,349.24,30.29,6.00),v60,z5,tPen\WObj:=wPaper;
    MoveL Offs(pOrigin,348.60,29.23,6.00),vTravel,z5,tPen\WObj:=wPaper;
    MoveL Offs(pOrigin,348.60,29.23,0.00),v60,z0,tPen\WObj:=wPaper;
    MoveL Offs(pOrigin,348.81,29.65,0.00),v40,z0,tPen\WObj:=wPaper;
    MoveL Offs(pOrigin,348.60,29.23,0.00),v40,fine,tPen\WObj:=wPaper;
    MoveL Offs(pOrigin,348.60,29.23,6.00),v60,z5,tPen\WObj:=wPaper;
    MoveL Offs(pOrigin,347.75,30.29,6.00),vTravel,z5,tPen\WObj:=wPaper;
    MoveL Offs(pOrigin,347.75,30.29,0.00),v60,z0,tPen\WObj:=wPaper;
    MoveL Offs(pOrigin,347.96,30.71,0.00),v40,z0,tPen\WObj:=wPaper;
    MoveL Offs(pOrigin,347.75,30.29,0.00),v40,fine,tPen\WObj:=wPaper;
    MoveL Offs(pOrigin,347.75,30.29,6.00),v60,z5,tPen\WObj:=wPaper;
    MoveL Offs(pOrigin,346.69,32.41,6.00),vTravel,z5,tPen\WObj:=wPaper;
    MoveL Offs(pOrigin,346.69,32.41,0.00),v60,z0,tPen\WObj:=wPaper;
    MoveL Offs(pOrigin,346.90,32.84,0.00),v40,z0,tPen\WObj:=wPaper;
    MoveL Offs(pOrigin,346.69,32.41,0.00),v40,fine,tPen\WObj:=wPaper;
    MoveL Offs(pOrigin,346.69,32.41,6.00),v60,z5,tPen\WObj:=wPaper;
    MoveL Offs(pOrigin,345.41,33.69,6.00),vTravel,z5,tPen\WObj:=wPaper;
    MoveL Offs(pOrigin,345.41,33.69,0.00),v60,z0,tPen\WObj:=wPaper;
    MoveL Offs(pOrigin,345.62,34.11,0.00),v40,z0,tPen\WObj:=wPaper;
    MoveL Offs(pOrigin,345.41,33.69,0.00),v40,fine,tPen\WObj:=wPaper;
    MoveL Offs(pOrigin,345.41,33.69,6.00),v60,z5,tPen\WObj:=wPaper;
    MoveL Offs(pOrigin,344.14,32.20,6.00),vTravel,z5,tPen\WObj:=wPaper;
    MoveL Offs(pOrigin,344.14,32.20,0.00),v60,z0,tPen\WObj:=wPaper;
    MoveL Offs(pOrigin,344.99,33.05,0.00),v40,z0,tPen\WObj:=wPaper;
    MoveL Offs(pOrigin,344.14,32.20,0.00),v40,fine,tPen\WObj:=wPaper;
    MoveL Offs(pOrigin,344.14,32.20,6.00),v60,z5,tPen\WObj:=wPaper;
    MoveL Offs(pOrigin,342.86,31.35,6.00),vTravel,z5,tPen\WObj:=wPaper;
    MoveL Offs(pOrigin,342.86,31.35,0.00),v60,z0,tPen\WObj:=wPaper;
    MoveL Offs(pOrigin,343.50,31.77,0.00),v40,z0,tPen\WObj:=wPaper;
    MoveL Offs(pOrigin,342.86,31.35,0.00),v40,z0,tPen\WObj:=wPaper;
    MoveL Offs(pOrigin,342.01,30.92,0.00),v40,z0,tPen\WObj:=wPaper;
    MoveL Offs(pOrigin,342.44,31.14,0.00),v40,z0,tPen\WObj:=wPaper;
    MoveL Offs(pOrigin,342.01,30.92,0.00),v40,fine,tPen\WObj:=wPaper;
    MoveL Offs(pOrigin,342.01,30.92,6.00),v60,z5,tPen\WObj:=wPaper;
    MoveL Offs(pOrigin,343.29,29.86,6.00),vTravel,z5,tPen\WObj:=wPaper;
    MoveL Offs(pOrigin,343.29,29.86,0.00),v60,z0,tPen\WObj:=wPaper;
    MoveL Offs(pOrigin,342.01,28.94,0.00),v40,z0,tPen\WObj:=wPaper;
    MoveL Offs(pOrigin,340.31,28.59,0.00),v40,fine,tPen\WObj:=wPaper;
    MoveL Offs(pOrigin,340.31,28.59,6.00),v60,z5,tPen\WObj:=wPaper;
    MoveL Offs(pOrigin,343.29,28.16,6.00),vTravel,z5,tPen\WObj:=wPaper;
    MoveL Offs(pOrigin,343.29,28.16,0.00),v60,z0,tPen\WObj:=wPaper;
    MoveL Offs(pOrigin,345.20,29.86,0.00),v40,z0,tPen\WObj:=wPaper;
    MoveL Offs(pOrigin,343.29,28.16,0.00),v40,fine,tPen\WObj:=wPaper;
    MoveL Offs(pOrigin,343.29,28.16,6.00),v60,z5,tPen\WObj:=wPaper;
    MoveL Offs(pOrigin,344.14,26.67,6.00),vTravel,z5,tPen\WObj:=wPaper;
    MoveL Offs(pOrigin,344.14,26.67,0.00),v60,z0,tPen\WObj:=wPaper;
    MoveL Offs(pOrigin,344.77,27.10,0.00),v40,z0,tPen\WObj:=wPaper;
    MoveL Offs(pOrigin,344.14,26.67,0.00),v40,fine,tPen\WObj:=wPaper;
  ENDPROC

